KUKA KRL program: EPS_2_251806_MH09A_A_20260223023037.src

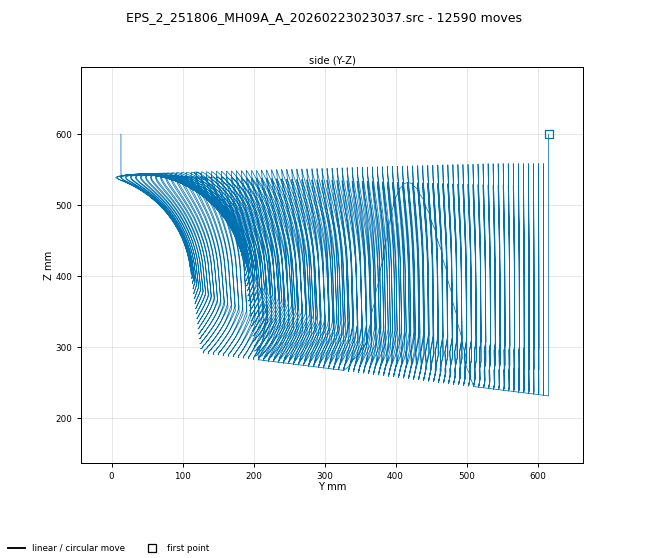
[picture p0: tool path of EPS_2_251806_MH09A_A_20260223023037.src, 12590 of 12592 moves have a stored position in this frame; points joined in program order, loops and branches not executed]
&ACCESS RVP
&REL 4
&COMMENT QRS 19112012
&PARAM EDITMASK = *
DEF PART()
EXT BAS (BAS_COMMAND :IN,REAL :IN )
INT I
BAS (#INITMOV,0 )

;KUKA QRS Post kuka4.cps  Date:22-06-2017 !

File_ID=3077

QRS_PRE_INIT()

;Init var - Until changes are made in qrs_pre_init
Outlet_Square_prg=0
Inlet_1_Square_prg=0
Inlet_2_Square_prg=0
Inlet_3_Square_prg=0
Inlet_4_Square_prg=0
Inlet_5_Square_prg=0

Outlet_1={X 0.000, Y 532.860, Z 433.000, B 0.000, E1 0.000 }
Inlet_1={X 0.000, Y 535.020, Z 403.000, B 0.000, E1 166.000 }
Outlet_1_type=251
Inlet_1_type=251
;QRS#1=Sidecore dimensions
;QRS#2=250-10" PVC SDR 35
;QRS#3=250-10" PVC SDR 35
;QRS#4=
;QRS#5=
;QRS#6=
;QRS#7=
;QRS#8=
;QRS#9=14M PSX
;QRS#10=14M PSX
;QRS#11=
;QRS#12=
;QRS#13=
;QRS#14=
;QRS#15=
;QRS#16=1220x127x838 2,75'
;QRS#17=EPS Height
;QRS#18=558,5
;QRS#19=*
;QRS#20= UPDATED VERSION 22-06-2017
;QRS#21=*
Outlet_Square=0100
Inlet_1_Square=0100
Inlet_2_Square=0
Inlet_3_Square=0
Inlet_4_Square=0
Inlet_5_Square=0
Mill_Square=1
Outlet_Square_Prg=205
Inlet_1_Square_prg=205

QRS_INIT()

$ADVANCE=5

; T1
PTP {E1 173.595,E2 173.595}
PTP {X 0,Y 615.506,A -85,B 0,C 180,E1 173.595,E2 173.595,E3 0,E4 0,E5 0,E6 0}
QRS_SPEED_INIT()
LIN {X 0,Y 615.506,Z 600,A -85,B 0,C 180,E1 173.595,E2 173.595,E3 0,E4 0,E5 0,E6 0} C_VEL
LIN {X 0,Y 615.506,Z 241.488,A -85,B 0,C 180,E1 173.595,E2 173.595} C_VEL
LIN {X 0,Y 615.506,Z 233.311,A -85,B 0,C 180,E1 173.595,E2 173.595} C_VEL
LIN {X 0,Y 615.49,Z 231.311,A -85,B 0,C 180,E1 173.408,E2 173.408} C_VEL
LIN {X 0,Y 615.485,Z 231.324,A -85,B 0,C 180,E1 170.802,E2 170.802} C_VEL
LIN {X 0,Y 615.466,Z 231.313,A -85,B 0,C 180,E1 168.14,E2 168.14} C_VEL
LIN {X 0,Y 615.489,Z 231.314,A -85,B 0,C 180,E1 165.452,E2 165.452} C_VEL
LIN {X 0,Y 615.469,Z 231.32,A -85,B 0,C 180,E1 162.73,E2 162.73} C_VEL
LIN {X 0,Y 615.486,Z 231.309,A -85,B 0,C 180,E1 159.968,E2 159.968} C_VEL
LIN {X 0,Y 615.488,Z 231.326,A -85,B 0,C 180,E1 157.157,E2 157.157} C_VEL
LIN {X 0,Y 615.46,Z 231.314,A -85,B 0,C 180,E1 154.434,E2 154.434} C_VEL
LIN {X 0,Y 615.49,Z 231.32,A -85,B 0,C 180,E1 151.547,E2 151.547} C_VEL
LIN {X 0,Y 615.462,Z 231.319,A -85,B 0,C 180,E1 148.916,E2 148.916} C_VEL
LIN {X 0,Y 615.464,Z 231.313,A -85,B 0,C 180,E1 146.467,E2 146.467} C_VEL
LIN {X 0,Y 615.485,Z 231.326,A -85,B 0,C 180,E1 143.577,E2 143.577} C_VEL
LIN {X 0,Y 615.456,Z 231.318,A -85,B 0,C 180,E1 140.94,E2 140.94} C_VEL
LIN {X 0,Y 615.467,Z 231.312,A -85,B 0,C 180,E1 138.526,E2 138.526} C_VEL
LIN {X 0,Y 615.494,Z 231.32,A -85,B 0,C 180,E1 135.853,E2 135.853} C_VEL
LIN {X 0,Y 615.458,Z 231.32,A -85,B 0,C 180,E1 133.246,E2 133.246} C_VEL
LIN {X 0,Y 615.47,Z 231.312,A -85,B 0,C 180,E1 130.607,E2 130.607} C_VEL
LIN {X 0,Y 615.49,Z 231.321,A -85,B 0,C 180,E1 128.015,E2 128.015} C_VEL
LIN {X 0,Y 615.467,Z 231.323,A -85,B 0,C 180,E1 125.616,E2 125.616} C_VEL
LIN {X 0,Y 615.48,Z 231.4,A -85,B 0,C 180,E1 124.594,E2 124.594} C_VEL
LIN {X 0,Y 615.442,Z 251.553,A -85,B 0,C 180,E1 121.687,E2 121.687} C_VEL
LIN {X 0,Y 615.455,Z 266.631,A -85,B 0,C 180,E1 119.539,E2 119.539} C_VEL
LIN {X 0,Y 615.471,Z 403.927,A -85,B 0,C 180,E1 117.892,E2 117.892} C_VEL
LIN {X 0,Y 615.484,Z 417.858,A -85,B 0,C 180,E1 117.591,E2 117.591} C_VEL
LIN {X 0,Y 615.487,Z 431.149,A -85,B 0,C 180,E1 117.176,E2 117.176} C_VEL
LIN {X 0,Y 615.488,Z 443.486,A -85,B 0,C 180,E1 116.67,E2 116.67} C_VEL
LIN {X 0,Y 615.485,Z 456.521,A -85,B 0,C 180,E1 115.988,E2 115.988} C_VEL
LIN {X 0,Y 615.497,Z 468.489,A -85,B 0,C 180,E1 115.209,E2 115.209} C_VEL
LIN {X 0,Y 615.499,Z 479.223,A -85,B 0,C 180,E1 114.361,E2 114.361} C_VEL
LIN {X 0,Y 615.497,Z 489.526,A -85,B 0,C 180,E1 113.377,E2 113.377} C_VEL
LIN {X 0,Y 615.492,Z 498.404,A -85,B 0,C 180,E1 112.351,E2 112.351} C_VEL
LIN {X 0,Y 615.494,Z 506.202,A -85,B 0,C 180,E1 111.255,E2 111.255} C_VEL
LIN {X 0,Y 615.495,Z 513.201,A -85,B 0,C 180,E1 110.032,E2 110.032} C_VEL
LIN {X 0,Y 615.492,Z 517.963,A -85,B 0,C 180,E1 108.991,E2 108.991} C_VEL
LIN {X 0,Y 615.495,Z 521.668,A -85,B 0,C 180,E1 107.956,E2 107.956} C_VEL
LIN {X 0,Y 615.493,Z 525.224,A -85,B 0,C 180,E1 106.586,E2 106.586} C_VEL
LIN {X 0,Y 615.493,Z 527.272,A -85,B 0,C 180,E1 105.225,E2 105.225} C_VEL
LIN {X 0,Y 615.497,Z 527.875,A -85,B 0,C 180,E1 103.874,E2 103.874} C_VEL
LIN {X 0,Y 615.489,Z 527.09,A -85,B 0,C 180,E1 102.53,E2 102.53} C_VEL
LIN {X 0,Y 615.491,Z 524.939,A -85,B 0,C 180,E1 101.193,E2 101.193} C_VEL
LIN {X 0,Y 615.499,Z 521.372,A -85,B 0,C 180,E1 99.862,E2 99.862} C_VEL
LIN {X 0,Y 615.494,Z 516.318,A -85,B 0,C 180,E1 98.536,E2 98.536} C_VEL
LIN {X 0,Y 615.495,Z 511.431,A -85,B 0,C 180,E1 97.545,E2 97.545} C_VEL
LIN {X 0,Y 615.497,Z 504.433,A -85,B 0,C 180,E1 96.392,E2 96.392} C_VEL
LIN {X 0,Y 615.497,Z 495.804,A -85,B 0,C 180,E1 95.241,E2 95.241} C_VEL
LIN {X 0,Y 615.497,Z 486.825,A -85,B 0,C 180,E1 94.256,E2 94.256} C_VEL
LIN {X 0,Y 615.497,Z 475.98,A -85,B 0,C 180,E1 93.273,E2 93.273} C_VEL
LIN {X 0,Y 615.498,Z 464.982,A -85,B 0,C 180,E1 92.454,E2 92.454} C_VEL
LIN {X 0,Y 615.491,Z 452.914,A -85,B 0,C 180,E1 91.718,E2 91.718} C_VEL
LIN {X 0,Y 615.494,Z 441.384,A -85,B 0,C 180,E1 91.145,E2 91.145} C_VEL
LIN {X 0,Y 615.492,Z 427.678,A -85,B 0,C 180,E1 90.613,E2 90.613} C_VEL
LIN {X 0,Y 615.47,Z 414.956,A -85,B 0,C 180,E1 90.245,E2 90.245} C_VEL
LIN {X 0,Y 615.453,Z 401.475,A -85,B 0,C 180,E1 89.979,E2 89.979} C_VEL
LIN {X 0,Y 615.447,Z 266.584,A -85,B 0,C 180,E1 88.364,E2 88.364} C_VEL
LIN {X 0,Y 615.484,Z 248.197,A -85,B 0,C 180,E1 85.744,E2 85.744} C_VEL
LIN {X 0,Y 615.489,Z 231.309,A -85,B 0,C 180,E1 83.293,E2 83.293} C_VEL
LIN {X 0,Y 615.476,Z 231.311,A -85,B 0,C 180,E1 80.801,E2 80.801} C_VEL
LIN {X 0,Y 615.487,Z 231.326,A -85,B 0,C 180,E1 78.139,E2 78.139} C_VEL
LIN {X 0,Y 615.484,Z 231.31,A -85,B 0,C 180,E1 75.451,E2 75.451} C_VEL
LIN {X 0,Y 615.472,Z 231.315,A -85,B 0,C 180,E1 72.729,E2 72.729} C_VEL
LIN {X 0,Y 615.485,Z 231.319,A -85,B 0,C 180,E1 69.968,E2 69.968} C_VEL
LIN {X 0,Y 615.479,Z 231.31,A -85,B 0,C 180,E1 67.156,E2 67.156} C_VEL
LIN {X 0,Y 615.496,Z 231.324,A -85,B 0,C 180,E1 64.285,E2 64.285} C_VEL
LIN {X 0,Y 615.483,Z 231.309,A -85,B 0,C 180,E1 61.342,E2 61.342} C_VEL
LIN {X 0,Y 615.474,Z 231.316,A -85,B 0,C 180,E1 58.913,E2 58.913} C_VEL
LIN {X 0,Y 615.498,Z 231.325,A -85,B 0,C 180,E1 56.462,E2 56.462} C_VEL
LIN {X 0,Y 615.485,Z 231.308,A -85,B 0,C 180,E1 53.576,E2 53.576} C_VEL
LIN {X 0,Y 615.477,Z 231.318,A -85,B 0,C 180,E1 50.937,E2 50.937} C_VEL
LIN {X 0,Y 615.493,Z 231.323,A -85,B 0,C 180,E1 48.528,E2 48.528} C_VEL
LIN {X 0,Y 615.492,Z 231.307,A -85,B 0,C 180,E1 45.852,E2 45.852} C_VEL
LIN {X 0,Y 615.479,Z 231.319,A -85,B 0,C 180,E1 43.048,E2 43.048} C_VEL
LIN {X 0,Y 615.483,Z 231.323,A -85,B 0,C 180,E1 40.605,E2 40.605} C_VEL
LIN {X 0,Y 615.484,Z 231.309,A -85,B 0,C 180,E1 38.013,E2 38.013} C_VEL
LIN {X 0,Y 615.479,Z 231.311,A -85,B 0,C 180,E1 35.615,E2 35.615} C_VEL
LIN {X 0,Y 615.479,Z 231.319,A -85,B 0,C 180,E1 33.235,E2 33.235} C_VEL
LIN {X 0,Y 615.489,Z 231.327,A -85,B 0,C 180,E1 30.918,E2 30.918} C_VEL
LIN {X 0,Y 615.479,Z 231.314,A -85,B 0,C 180,E1 28.451,E2 28.451} C_VEL
LIN {X 0,Y 615.478,Z 231.312,A -85,B 0,C 180,E1 25.715,E2 25.715} C_VEL
LIN {X 0,Y 615.475,Z 231.316,A -85,B 0,C 180,E1 23.556,E2 23.556} C_VEL
LIN {X 0,Y 615.479,Z 231.319,A -85,B 0,C 180,E1 21.431,E2 21.431} C_VEL
LIN {X 0,Y 615.477,Z 231.314,A -85,B 0,C 180,E1 18.605,E2 18.605} C_VEL
LIN {X 0,Y 615.476,Z 231.312,A -85,B 0,C 180,E1 15.904,E2 15.904} C_VEL
LIN {X 0,Y 615.494,Z 231.324,A -85,B 0,C 180,E1 13.2,E2 13.2} C_VEL
LIN {X 0,Y 615.486,Z 231.309,A -85,B 0,C 180,E1 10.526,E2 10.526} C_VEL
LIN {X 0,Y 615.477,Z 231.315,A -85,B 0,C 180,E1 7.875,E2 7.875} C_VEL
LIN {X 0,Y 615.487,Z 231.322,A -85,B 0,C 180,E1 5.24,E2 5.24} C_VEL
LIN {X 0,Y 615.488,Z 231.308,A -85,B 0,C 180,E1 2.617,E2 2.617} C_VEL
LIN {X 0,Y 615.478,Z 231.315,A -85,B 0,C 180,E1 -0.001,E2 -0.001} C_VEL
LIN {X 0,Y 615.486,Z 231.322,A -85,B 0,C 180,E1 -2.619,E2 -2.619} C_VEL
LIN {X 0,Y 615.487,Z 231.308,A -85,B 0,C 180,E1 -5.242,E2 -5.242} C_VEL
LIN {X 0,Y 615.479,Z 231.315,A -85,B 0,C 180,E1 -7.877,E2 -7.877} C_VEL
LIN {X 0,Y 615.484,Z 231.321,A -85,B 0,C 180,E1 -10.528,E2 -10.528} C_VEL
LIN {X 0,Y 615.493,Z 231.306,A -85,B 0,C 180,E1 -13.202,E2 -13.202} C_VEL
LIN {X 0,Y 615.482,Z 231.319,A -85,B 0,C 180,E1 -15.906,E2 -15.906} C_VEL
LIN {X 0,Y 615.475,Z 231.316,A -85,B 0,C 180,E1 -18.647,E2 -18.647} C_VEL
LIN {X 0,Y 615.479,Z 231.312,A -85,B 0,C 180,E1 -21.433,E2 -21.433} C_VEL
LIN {X 0,Y 615.483,Z 231.321,A -85,B 0,C 180,E1 -24.273,E2 -24.273} C_VEL
LIN {X 0,Y 615.491,Z 231.307,A -85,B 0,C 180,E1 -27.178,E2 -27.178} C_VEL
LIN {X 0,Y 615.483,Z 231.321,A -85,B 0,C 180,E1 -30.161,E2 -30.161} C_VEL
LIN {X 0,Y 615.473,Z 231.315,A -85,B 0,C 180,E1 -32.459,E2 -32.459} C_VEL
LIN {X 0,Y 615.49,Z 231.307,A -85,B 0,C 180,E1 -34.815,E2 -34.815} C_VEL
LIN {X 0,Y 615.482,Z 231.313,A -85,B 0,C 180,E1 -37.243,E2 -37.243} C_VEL
LIN {X 0,Y 615.474,Z 231.32,A -85,B 0,C 180,E1 -40.089,E2 -40.089} C_VEL
LIN {X 0,Y 615.473,Z 231.313,A -85,B 0,C 180,E1 -42.355,E2 -42.355} C_VEL
LIN {X 0,Y 615.483,Z 231.312,A -85,B 0,C 180,E1 -45.069,E2 -45.069} C_VEL
LIN {X 0,Y 615.496,Z 231.325,A -85,B 0,C 180,E1 -47.649,E2 -47.649} C_VEL
LIN {X 0,Y 615.474,Z 231.313,A -85,B 0,C 180,E1 -50.25,E2 -50.25} C_VEL
LIN {X 0,Y 615.479,Z 231.315,A -85,B 0,C 180,E1 -53.065,E2 -53.065} C_VEL
LIN {X 0,Y 615.489,Z 231.321,A -85,B 0,C 180,E1 -55.3,E2 -55.3} C_VEL
LIN {X 0,Y 615.482,Z 231.321,A -85,B 0,C 180,E1 -57.671,E2 -57.671} C_VEL
LIN {X 0,Y 615.493,Z 231.307,A -85,B 0,C 180,E1 -60.595,E2 -60.595} C_VEL
LIN {X 0,Y 615.48,Z 231.321,A -85,B 0,C 180,E1 -63.556,E2 -63.556} C_VEL
LIN {X 0,Y 615.486,Z 231.309,A -85,B 0,C 180,E1 -66.444,E2 -66.444} C_VEL
LIN {X 0,Y 615.486,Z 231.548,A -85,B 0,C 180,E1 -66.533,E2 -66.533} C_VEL
LIN {X 0,Y 615.487,Z 254.856,A -85,B 0,C 180,E1 -69.444,E2 -69.444} C_VEL
LIN {X 0,Y 615.493,Z 277.448,A -85,B 0,C 180,E1 -72.215,E2 -72.215} C_VEL
LIN {X 0,Y 615.49,Z 295.428,A -85,B 0,C 180,E1 -74.393,E2 -74.393} C_VEL
LIN {X 0,Y 615.488,Z 433.076,A -85,B 0,C 180,E1 -76.048,E2 -76.048} C_VEL
LIN {X 0,Y 615.494,Z 446.865,A -85,B 0,C 180,E1 -76.337,E2 -76.337} C_VEL
LIN {X 0,Y 615.487,Z 460.574,A -85,B 0,C 180,E1 -76.757,E2 -76.757} C_VEL
LIN {X 0,Y 615.497,Z 473.841,A -85,B 0,C 180,E1 -77.303,E2 -77.303} C_VEL
LIN {X 0,Y 615.483,Z 486.604,A -85,B 0,C 180,E1 -77.972,E2 -77.972} C_VEL
LIN {X 0,Y 615.499,Z 499.342,A -85,B 0,C 180,E1 -78.807,E2 -78.807} C_VEL
LIN {X 0,Y 615.498,Z 509.75,A -85,B 0,C 180,E1 -79.64,E2 -79.64} C_VEL
LIN {X 0,Y 615.496,Z 520.089,A -85,B 0,C 180,E1 -80.636,E2 -80.636} C_VEL
LIN {X 0,Y 615.497,Z 528.603,A -85,B 0,C 180,E1 -81.629,E2 -81.629} C_VEL
LIN {X 0,Y 615.496,Z 536.727,A -85,B 0,C 180,E1 -82.785,E2 -82.785} C_VEL
LIN {X 0,Y 615.496,Z 542.43,A -85,B 0,C 180,E1 -83.773,E2 -83.773} C_VEL
LIN {X 0,Y 615.495,Z 547.08,A -85,B 0,C 180,E1 -84.759,E2 -84.759} C_VEL
LIN {X 0,Y 615.494,Z 551.902,A -85,B 0,C 180,E1 -86.072,E2 -86.072} C_VEL
LIN {X 0,Y 615.496,Z 555.252,A -85,B 0,C 180,E1 -87.382,E2 -87.382} C_VEL
LIN {X 0,Y 615.489,Z 557.229,A -85,B 0,C 180,E1 -88.691,E2 -88.691} C_VEL
LIN {X 0,Y 615.493,Z 557.889,A -85,B 0,C 180,E1 -90,E2 -90} C_VEL
LIN {X 0,Y 615.489,Z 557.229,A -85,B 0,C 180,E1 -91.308,E2 -91.308} C_VEL
LIN {X 0,Y 615.496,Z 555.252,A -85,B 0,C 180,E1 -92.618,E2 -92.618} C_VEL
LIN {X 0,Y 615.494,Z 551.902,A -85,B 0,C 180,E1 -93.928,E2 -93.928} C_VEL
LIN {X 0,Y 615.495,Z 547.081,A -85,B 0,C 180,E1 -95.241,E2 -95.241} C_VEL
LIN {X 0,Y 615.496,Z 540.629,A -85,B 0,C 180,E1 -96.556,E2 -96.556} C_VEL
LIN {X 0,Y 615.497,Z 533.442,A -85,B 0,C 180,E1 -97.71,E2 -97.71} C_VEL
LIN {X 0,Y 615.498,Z 525.905,A -85,B 0,C 180,E1 -98.702,E2 -98.702} C_VEL
LIN {X 0,Y 615.496,Z 516.855,A -85,B 0,C 180,E1 -99.696,E2 -99.696} C_VEL
LIN {X 0,Y 615.498,Z 506.76,A -85,B 0,C 180,E1 -100.618,E2 -100.618} C_VEL
LIN {X 0,Y 615.498,Z 495.862,A -85,B 0,C 180,E1 -101.443,E2 -101.443} C_VEL
LIN {X 0,Y 615.484,Z 483.712,A -85,B 0,C 180,E1 -102.195,E2 -102.195} C_VEL
LIN {X 0,Y 615.493,Z 470.098,A -85,B 0,C 180,E1 -102.865,E2 -102.865} C_VEL
LIN {X 0,Y 615.49,Z 456.845,A -85,B 0,C 180,E1 -103.369,E2 -103.369} C_VEL
LIN {X 0,Y 615.493,Z 443.301,A -85,B 0,C 180,E1 -103.747,E2 -103.747} C_VEL
LIN {X 0,Y 615.485,Z 428.996,A -85,B 0,C 180,E1 -104.009,E2 -104.009} C_VEL
LIN {X 0,Y 615.49,Z 295.43,A -85,B 0,C 180,E1 -105.607,E2 -105.607} C_VEL
LIN {X 0,Y 615.483,Z 273.41,A -85,B 0,C 180,E1 -108.277,E2 -108.277} C_VEL
LIN {X 0,Y 615.469,Z 252.038,A -85,B 0,C 180,E1 -110.906,E2 -110.906} C_VEL
LIN {X 0,Y 615.485,Z 231.309,A -85,B 0,C 180,E1 -113.511,E2 -113.511} C_VEL
LIN {X 0,Y 615.485,Z 231.308,A -85,B 0,C 180,E1 -115.715,E2 -115.715} C_VEL
LIN {X 0,Y 615.485,Z 231.327,A -85,B 0,C 180,E1 -118.657,E2 -118.657} C_VEL
LIN {X 0,Y 615.481,Z 231.314,A -85,B 0,C 180,E1 -121.085,E2 -121.085} C_VEL
LIN {X 0,Y 615.492,Z 231.307,A -85,B 0,C 180,E1 -123.534,E2 -123.534} C_VEL
LIN {X 0,Y 615.484,Z 231.328,A -85,B 0,C 180,E1 -126.424,E2 -126.424} C_VEL
LIN {X 0,Y 615.483,Z 231.311,A -85,B 0,C 180,E1 -129.061,E2 -129.061} C_VEL
LIN {X 0,Y 615.486,Z 231.308,A -85,B 0,C 180,E1 -131.473,E2 -131.473} C_VEL
LIN {X 0,Y 615.49,Z 231.323,A -85,B 0,C 180,E1 -134.148,E2 -134.148} C_VEL
LIN {X 0,Y 615.483,Z 231.31,A -85,B 0,C 180,E1 -136.952,E2 -136.952} C_VEL
LIN {X 0,Y 615.482,Z 231.31,A -85,B 0,C 180,E1 -139.393,E2 -139.393} C_VEL
LIN {X 0,Y 615.483,Z 231.324,A -85,B 0,C 180,E1 -141.987,E2 -141.987} C_VEL
LIN {X 0,Y 615.479,Z 231.319,A -85,B 0,C 180,E1 -144.383,E2 -144.383} C_VEL
LIN {X 0,Y 615.48,Z 231.31,A -85,B 0,C 180,E1 -146.763,E2 -146.763} C_VEL
LIN {X 0,Y 615.487,Z 231.308,A -85,B 0,C 180,E1 -149.08,E2 -149.08} C_VEL
LIN {X 0,Y 615.48,Z 231.318,A -85,B 0,C 180,E1 -151.549,E2 -151.549} C_VEL
LIN {X 0,Y 615.473,Z 231.317,A -85,B 0,C 180,E1 -154.283,E2 -154.283} C_VEL
LIN {X 0,Y 615.472,Z 231.314,A -85,B 0,C 180,E1 -156.442,E2 -156.442} C_VEL
LIN {X 0,Y 615.483,Z 231.315,A -85,B 0,C 180,E1 -159.268,E2 -159.268} C_VEL
LIN {X 0,Y 615.475,Z 231.319,A -85,B 0,C 180,E1 -162.042,E2 -162.042} C_VEL
LIN {X 0,Y 615.49,Z 231.308,A -85,B 0,C 180,E1 -164.773,E2 -164.773} C_VEL
LIN {X 0,Y 615.486,Z 231.325,A -85,B 0,C 180,E1 -167.469,E2 -167.469} C_VEL
LIN {X 0,Y 615.47,Z 231.314,A -85,B 0,C 180,E1 -170.137,E2 -170.137} C_VEL
LIN {X 0,Y 615.487,Z 231.31,A -85,B 0,C 180,E1 -172.784,E2 -172.784} C_VEL
LIN {X 0,Y 615.496,Z 231.325,A -85,B 0,C 180,E1 -175.415,E2 -175.415} C_VEL
LIN {X 0,Y 615.468,Z 231.314,A -85,B 0,C 180,E1 -178.036,E2 -178.036} C_VEL
LIN {X 0,Y 615.486,Z 231.311,A -85,B 0,C 180,E1 -180.653,E2 -180.653} C_VEL
LIN {X 0,Y 615.488,Z 231.325,A -85,B 0,C 180,E1 -183.272,E2 -183.272} C_VEL
LIN {X 0,Y 615.466,Z 231.314,A -85,B 0,C 180,E1 -185.898,E2 -185.898} C_VEL
LIN {X 0,Y 615.49,Z 231.311,A -85,B 0,C 180,E1 -186.592,E2 -186.592} C_VEL
LIN {X 0,Y 614.813,Z 231.47,A -85,B 0,C 180,E1 -187.138,E2 -187.138} C_VEL
LIN {X 0,Y 611.977,Z 231.873,A -85,B 0,C 180,E1 -188.024,E2 -188.024} C_VEL
LIN {X 0,Y 609.583,Z 232.188,A -85,B 0,C 180,E1 -188.736,E2 -188.736} C_VEL
LIN {X 0,Y 608.543,Z 232.308,A -85,B 0,C 180,E1 -189.286,E2 -189.286} C_VEL
LIN {X 0,Y 608.451,Z 232.317,A -85,B 0,C 180,E1 -189.472,E2 -189.472} C_VEL
LIN {X 0,Y 608.447,Z 232.313,A -85,B 0,C 180,E1 -191.999,E2 -191.999} C_VEL
LIN {X 0,Y 608.472,Z 232.316,A -85,B 0,C 180,E1 -194.719,E2 -194.719} C_VEL
LIN {X 0,Y 608.437,Z 232.316,A -85,B 0,C 180,E1 -197.476,E2 -197.476} C_VEL
LIN {X 0,Y 608.462,Z 232.313,A -85,B 0,C 180,E1 -200.273,E2 -200.273} C_VEL
LIN {X 0,Y 608.441,Z 232.319,A -85,B 0,C 180,E1 -203.123,E2 -203.123} C_VEL
LIN {X 0,Y 608.451,Z 232.313,A -85,B 0,C 180,E1 -205.72,E2 -205.72} C_VEL
LIN {X 0,Y 608.473,Z 232.32,A -85,B 0,C 180,E1 -208.622,E2 -208.622} C_VEL
LIN {X 0,Y 608.429,Z 232.316,A -85,B 0,C 180,E1 -211.317,E2 -211.317} C_VEL
LIN {X 0,Y 608.459,Z 232.312,A -85,B 0,C 180,E1 -213.735,E2 -213.735} C_VEL
LIN {X 0,Y 608.467,Z 232.314,A -85,B 0,C 180,E1 -216.089,E2 -216.089} C_VEL
LIN {X 0,Y 608.454,Z 232.32,A -85,B 0,C 180,E1 -218.587,E2 -218.587} C_VEL
LIN {X 0,Y 608.438,Z 232.314,A -85,B 0,C 180,E1 -221.341,E2 -221.341} C_VEL
LIN {X 0,Y 608.47,Z 232.314,A -85,B 0,C 180,E1 -223.867,E2 -223.867} C_VEL
LIN {X 0,Y 608.448,Z 232.317,A -85,B 0,C 180,E1 -226.691,E2 -226.691} C_VEL
LIN {X 0,Y 608.425,Z 232.318,A -85,B 0,C 180,E1 -228.822,E2 -228.822} C_VEL
LIN {X 0,Y 608.451,Z 232.314,A -85,B 0,C 180,E1 -231.412,E2 -231.412} C_VEL
LIN {X 0,Y 608.468,Z 232.319,A -85,B 0,C 180,E1 -233.949,E2 -233.949} C_VEL
LIN {X 0,Y 608.485,Z 232.486,A -85,B 0,C 180,E1 -235.316,E2 -235.316} C_VEL
LIN {X 0,Y 608.489,Z 250.245,A -85,B 0,C 180,E1 -237.908,E2 -237.908} C_VEL
LIN {X 0,Y 608.446,Z 266.656,A -85,B 0,C 180,E1 -240.268,E2 -240.268} C_VEL
LIN {X 0,Y 608.63,Z 273.911,A -85,B 0,C 180,E1 -240.373,E2 -240.373} C_VEL
LIN {X 0,Y 608.6,Z 402.894,A -85,B 0,C 180,E1 -241.929,E2 -241.929} C_VEL
LIN {X 0,Y 608.572,Z 417.186,A -85,B 0,C 180,E1 -242.232,E2 -242.232} C_VEL
LIN {X 0,Y 608.573,Z 431.379,A -85,B 0,C 180,E1 -242.679,E2 -242.679} C_VEL
LIN {X 0,Y 608.544,Z 444.524,A -85,B 0,C 180,E1 -243.231,E2 -243.231} C_VEL
LIN {X 0,Y 608.53,Z 456.673,A -85,B 0,C 180,E1 -243.877,E2 -243.877} C_VEL
LIN {X 0,Y 608.498,Z 469.197,A -85,B 0,C 180,E1 -244.702,E2 -244.702} C_VEL
LIN {X 0,Y 608.486,Z 479.815,A -85,B 0,C 180,E1 -245.554,E2 -245.554} C_VEL
LIN {X 0,Y 608.483,Z 489.811,A -85,B 0,C 180,E1 -246.518,E2 -246.518} C_VEL
LIN {X 0,Y 608.46,Z 499.058,A -85,B 0,C 180,E1 -247.595,E2 -247.595} C_VEL
LIN {X 0,Y 608.459,Z 506.609,A -85,B 0,C 180,E1 -248.664,E2 -248.664} C_VEL
LIN {X 0,Y 608.441,Z 512.759,A -85,B 0,C 180,E1 -249.726,E2 -249.726} C_VEL
LIN {X 0,Y 608.434,Z 517.727,A -85,B 0,C 180,E1 -250.78,E2 -250.78} C_VEL
LIN {X 0,Y 608.448,Z 522.778,A -85,B 0,C 180,E1 -252.177,E2 -252.177} C_VEL
LIN {X 0,Y 608.419,Z 526.013,A -85,B 0,C 180,E1 -253.481,E2 -253.481} C_VEL
LIN {X 0,Y 608.415,Z 527.679,A -85,B 0,C 180,E1 -254.593,E2 -254.593} C_VEL
LIN {X 0,Y 608.428,Z 528.494,A -85,B 0,C 180,E1 -255.992,E2 -255.992} C_VEL
LIN {X 0,Y 608.414,Z 527.884,A -85,B 0,C 180,E1 -257.322,E2 -257.322} C_VEL
LIN {X 0,Y 608.417,Z 525.87,A -85,B 0,C 180,E1 -258.675,E2 -258.675} C_VEL
LIN {X 0,Y 608.433,Z 522.43,A -85,B 0,C 180,E1 -260.023,E2 -260.023} C_VEL
LIN {X 0,Y 608.426,Z 517.496,A -85,B 0,C 180,E1 -261.364,E2 -261.364} C_VEL
LIN {X 0,Y 608.445,Z 512.745,A -85,B 0,C 180,E1 -262.367,E2 -262.367} C_VEL
LIN {X 0,Y 608.455,Z 505.374,A -85,B 0,C 180,E1 -263.61,E2 -263.61} C_VEL
LIN {X 0,Y 608.461,Z 497.416,A -85,B 0,C 180,E1 -264.698,E2 -264.698} C_VEL
LIN {X 0,Y 608.48,Z 488.625,A -85,B 0,C 180,E1 -265.695,E2 -265.695} C_VEL
LIN {X 0,Y 608.491,Z 478.048,A -85,B 0,C 180,E1 -266.69,E2 -266.69} C_VEL
LIN {X 0,Y 608.514,Z 466.264,A -85,B 0,C 180,E1 -267.601,E2 -267.601} C_VEL
LIN {X 0,Y 608.526,Z 454.439,A -85,B 0,C 180,E1 -268.346,E2 -268.346} C_VEL
LIN {X 0,Y 608.558,Z 441.332,A -85,B 0,C 180,E1 -269.008,E2 -269.008} C_VEL
LIN {X 0,Y 608.575,Z 427.573,A -85,B 0,C 180,E1 -269.545,E2 -269.545} C_VEL
LIN {X 0,Y 608.588,Z 413.878,A -85,B 0,C 180,E1 -269.938,E2 -269.938} C_VEL
LIN {X 0,Y 608.581,Z 399.69,A -85,B 0,C 180,E1 -270.207,E2 -270.207} C_VEL
LIN {X 0,Y 608.518,Z 267.308,A -85,B 0,C 180,E1 -271.799,E2 -271.799} C_VEL
LIN {X 0,Y 608.44,Z 266.67,A -85,B 0,C 180,E1 -271.82,E2 -271.82} C_VEL
LIN {X 0,Y 608.519,Z 248.244,A -85,B 0,C 180,E1 -274.471,E2 -274.471} C_VEL
LIN {X 0,Y 608.484,Z 232.31,A -85,B 0,C 180,E1 -276.805,E2 -276.805} C_VEL
LIN {X 0,Y 608.461,Z 232.313,A -85,B 0,C 180,E1 -279.306,E2 -279.306} C_VEL
LIN {X 0,Y 608.46,Z 232.321,A -85,B 0,C 180,E1 -282,E2 -282} C_VEL
LIN {X 0,Y 608.468,Z 232.311,A -85,B 0,C 180,E1 -284.72,E2 -284.72} C_VEL
LIN {X 0,Y 608.444,Z 232.318,A -85,B 0,C 180,E1 -287.477,E2 -287.477} C_VEL
LIN {X 0,Y 608.461,Z 232.314,A -85,B 0,C 180,E1 -290.274,E2 -290.274} C_VEL
LIN {X 0,Y 608.444,Z 232.315,A -85,B 0,C 180,E1 -293.124,E2 -293.124} C_VEL
LIN {X 0,Y 608.475,Z 232.319,A -85,B 0,C 180,E1 -295.725,E2 -295.725} C_VEL
LIN {X 0,Y 608.471,Z 232.31,A -85,B 0,C 180,E1 -298.623,E2 -298.623} C_VEL
LIN {X 0,Y 608.465,Z 232.317,A -85,B 0,C 180,E1 -301.316,E2 -301.316} C_VEL
LIN {X 0,Y 608.477,Z 232.316,A -85,B 0,C 180,E1 -303.738,E2 -303.738} C_VEL
LIN {X 0,Y 608.466,Z 232.312,A -85,B 0,C 180,E1 -306.09,E2 -306.09} C_VEL
LIN {X 0,Y 608.459,Z 232.312,A -85,B 0,C 180,E1 -308.588,E2 -308.588} C_VEL
LIN {X 0,Y 608.462,Z 232.322,A -85,B 0,C 180,E1 -311.344,E2 -311.344} C_VEL
LIN {X 0,Y 608.457,Z 232.312,A -85,B 0,C 180,E1 -314.266,E2 -314.266} C_VEL
LIN {X 0,Y 608.446,Z 232.32,A -85,B 0,C 180,E1 -317.041,E2 -317.041} C_VEL
LIN {X 0,Y 608.448,Z 232.316,A -85,B 0,C 180,E1 -319.698,E2 -319.698} C_VEL
LIN {X 0,Y 608.464,Z 232.311,A -85,B 0,C 180,E1 -322.255,E2 -322.255} C_VEL
LIN {X 0,Y 608.481,Z 232.319,A -85,B 0,C 180,E1 -325.089,E2 -325.089} C_VEL
LIN {X 0,Y 608.458,Z 232.312,A -85,B 0,C 180,E1 -327.907,E2 -327.907} C_VEL
LIN {X 0,Y 608.468,Z 232.311,A -85,B 0,C 180,E1 -330.222,E2 -330.222} C_VEL
LIN {X 0,Y 608.479,Z 232.316,A -85,B 0,C 180,E1 -332.79,E2 -332.79} C_VEL
LIN {X 0,Y 608.481,Z 232.309,A -85,B 0,C 180,E1 -335.844,E2 -335.844} C_VEL
LIN {X 0,Y 608.466,Z 232.313,A -85,B 0,C 180,E1 -338.31,E2 -338.31} C_VEL
LIN {X 0,Y 608.447,Z 232.319,A -85,B 0,C 180,E1 -341.131,E2 -341.131} C_VEL
LIN {X 0,Y 608.454,Z 232.312,A -85,B 0,C 180,E1 -343.907,E2 -343.907} C_VEL
LIN {X 0,Y 608.467,Z 232.32,A -85,B 0,C 180,E1 -346.645,E2 -346.645} C_VEL
LIN {X 0,Y 608.461,Z 232.313,A -85,B 0,C 180,E1 -349.351,E2 -349.351} C_VEL
LIN {X 0,Y 608.469,Z 232.312,A -85,B 0,C 180,E1 -352.034,E2 -352.034} C_VEL
LIN {X 0,Y 608.465,Z 232.32,A -85,B 0,C 180,E1 -354.699,E2 -354.699} C_VEL
LIN {X 0,Y 608.478,Z 232.31,A -85,B 0,C 180,E1 -357.353,E2 -357.353} C_VEL
LIN {X 0,Y 608.469,Z 232.313,A -85,B 0,C 180,E1 -360.001,E2 -360.001} C_VEL
LIN {X 0,Y 608.477,Z 232.316,A -85,B 0,C 180,E1 -362.649,E2 -362.649} C_VEL
LIN {X 0,Y 608.465,Z 232.311,A -85,B 0,C 180,E1 -365.303,E2 -365.303} C_VEL
LIN {X 0,Y 608.47,Z 232.314,A -85,B 0,C 180,E1 -367.968,E2 -367.968} C_VEL
LIN {X 0,Y 608.46,Z 232.316,A -85,B 0,C 180,E1 -370.651,E2 -370.651} C_VEL
LIN {X 0,Y 608.467,Z 232.311,A -85,B 0,C 180,E1 -373.357,E2 -373.357} C_VEL
LIN {X 0,Y 608.457,Z 232.321,A -85,B 0,C 180,E1 -376.095,E2 -376.095} C_VEL
LIN {X 0,Y 608.449,Z 232.314,A -85,B 0,C 180,E1 -378.87,E2 -378.87} C_VEL
LIN {X 0,Y 608.468,Z 232.314,A -85,B 0,C 180,E1 -381.692,E2 -381.692} C_VEL
LIN {X 0,Y 608.453,Z 232.315,A -85,B 0,C 180,E1 -384.572,E2 -384.572} C_VEL
LIN {X 0,Y 608.483,Z 232.309,A -85,B 0,C 180,E1 -387.21,E2 -387.21} C_VEL
LIN {X 0,Y 608.468,Z 232.321,A -85,B 0,C 180,E1 -389.974,E2 -389.974} C_VEL
LIN {X 0,Y 608.45,Z 232.314,A -85,B 0,C 180,E1 -392.522,E2 -392.522} C_VEL
LIN {X 0,Y 608.443,Z 232.316,A -85,B 0,C 180,E1 -395.278,E2 -395.278} C_VEL
LIN {X 0,Y 608.466,Z 232.321,A -85,B 0,C 180,E1 -397.747,E2 -397.747} C_VEL
LIN {X 0,Y 608.442,Z 232.316,A -85,B 0,C 180,E1 -400.329,E2 -400.329} C_VEL
LIN {X 0,Y 608.469,Z 232.314,A -85,B 0,C 180,E1 -403.31,E2 -403.31} C_VEL
LIN {X 0,Y 608.464,Z 232.314,A -85,B 0,C 180,E1 -406.131,E2 -406.131} C_VEL
LIN {X 0,Y 608.456,Z 232.312,A -85,B 0,C 180,E1 -408.825,E2 -408.825} C_VEL
LIN {X 0,Y 608.459,Z 232.318,A -85,B 0,C 180,E1 -411.761,E2 -411.761} C_VEL
LIN {X 0,Y 608.443,Z 232.317,A -85,B 0,C 180,E1 -413.955,E2 -413.955} C_VEL
LIN {X 0,Y 608.463,Z 232.311,A -85,B 0,C 180,E1 -416.33,E2 -416.33} C_VEL
LIN {X 0,Y 608.447,Z 232.314,A -85,B 0,C 180,E1 -418.733,E2 -418.733} C_VEL
LIN {X 0,Y 608.472,Z 232.321,A -85,B 0,C 180,E1 -421.381,E2 -421.381} C_VEL
LIN {X 0,Y 608.474,Z 232.31,A -85,B 0,C 180,E1 -424.279,E2 -424.279} C_VEL
LIN {X 0,Y 608.485,Z 232.431,A -85,B 0,C 180,E1 -426.36,E2 -426.36} C_VEL
LIN {X 0,Y 608.589,Z 249.21,A -85,B 0,C 180,E1 -428.491,E2 -428.491} C_VEL
LIN {X 0,Y 608.533,Z 271.49,A -85,B 0,C 180,E1 -431.267,E2 -431.267} C_VEL
LIN {X 0,Y 608.521,Z 294.428,A -85,B 0,C 180,E1 -434.08,E2 -434.08} C_VEL
LIN {X 0,Y 608.515,Z 295.576,A -85,B 0,C 180,E1 -434.22,E2 -434.22} C_VEL
LIN {X 0,Y 608.6,Z 433.465,A -85,B 0,C 180,E1 -435.894,E2 -435.894} C_VEL
LIN {X 0,Y 608.592,Z 447.633,A -85,B 0,C 180,E1 -436.2,E2 -436.2} C_VEL
LIN {X 0,Y 608.578,Z 461.716,A -85,B 0,C 180,E1 -436.646,E2 -436.646} C_VEL
LIN {X 0,Y 608.561,Z 473.887,A -85,B 0,C 180,E1 -437.155,E2 -437.155} C_VEL
LIN {X 0,Y 608.511,Z 486.683,A -85,B 0,C 180,E1 -437.832,E2 -437.832} C_VEL
LIN {X 0,Y 608.499,Z 499.473,A -85,B 0,C 180,E1 -438.677,E2 -438.677} C_VEL
LIN {X 0,Y 608.496,Z 509.933,A -85,B 0,C 180,E1 -439.519,E2 -439.519} C_VEL
LIN {X 0,Y 608.479,Z 520.335,A -85,B 0,C 180,E1 -440.527,E2 -440.527} C_VEL
LIN {X 0,Y 608.464,Z 528.915,A -85,B 0,C 180,E1 -441.532,E2 -441.532} C_VEL
LIN {X 0,Y 608.461,Z 537.114,A -85,B 0,C 180,E1 -442.701,E2 -442.701} C_VEL
LIN {X 0,Y 608.444,Z 543.546,A -85,B 0,C 180,E1 -443.831,E2 -443.831} C_VEL
LIN {X 0,Y 608.437,Z 548.962,A -85,B 0,C 180,E1 -445.03,E2 -445.03} C_VEL
LIN {X 0,Y 608.431,Z 552.441,A -85,B 0,C 180,E1 -446.026,E2 -446.026} C_VEL
LIN {X 0,Y 608.424,Z 555.831,A -85,B 0,C 180,E1 -447.352,E2 -447.352} C_VEL
LIN {X 0,Y 608.442,Z 557.83,A -85,B 0,C 180,E1 -448.676,E2 -448.676} C_VEL
LIN {X 0,Y 608.433,Z 558.5,A -85,B 0,C 180,E1 -450,E2 -450} C_VEL
LIN {X 0,Y 608.442,Z 557.831,A -85,B 0,C 180,E1 -451.324,E2 -451.324} C_VEL
LIN {X 0,Y 608.424,Z 555.831,A -85,B 0,C 180,E1 -452.648,E2 -452.648} C_VEL
LIN {X 0,Y 608.431,Z 552.442,A -85,B 0,C 180,E1 -453.974,E2 -453.974} C_VEL
LIN {X 0,Y 608.44,Z 547.568,A -85,B 0,C 180,E1 -455.302,E2 -455.302} C_VEL
LIN {X 0,Y 608.445,Z 541.212,A -85,B 0,C 180,E1 -456.603,E2 -456.603} C_VEL
LIN {X 0,Y 608.453,Z 533.799,A -85,B 0,C 180,E1 -457.8,E2 -457.8} C_VEL
LIN {X 0,Y 608.473,Z 524.825,A -85,B 0,C 180,E1 -458.97,E2 -458.97} C_VEL
LIN {X 0,Y 608.473,Z 515.394,A -85,B 0,C 180,E1 -459.977,E2 -459.977} C_VEL
LIN {X 0,Y 608.506,Z 504.049,A -85,B 0,C 180,E1 -460.973,E2 -460.973} C_VEL
LIN {X 0,Y 608.53,Z 492.153,A -85,B 0,C 180,E1 -461.829,E2 -461.829} C_VEL
LIN {X 0,Y 608.53,Z 479.078,A -85,B 0,C 180,E1 -462.591,E2 -462.591} C_VEL
LIN {X 0,Y 608.553,Z 466.18,A -85,B 0,C 180,E1 -463.184,E2 -463.184} C_VEL
LIN {X 0,Y 608.593,Z 452.193,A -85,B 0,C 180,E1 -463.672,E2 -463.672} C_VEL
LIN {X 0,Y 608.622,Z 438.471,A -85,B 0,C 180,E1 -464.012,E2 -464.012} C_VEL
LIN {X 0,Y 608.619,Z 422.194,A -85,B 0,C 180,E1 -464.257,E2 -464.257} C_VEL
LIN {X 0,Y 608.528,Z 295.577,A -85,B 0,C 180,E1 -465.78,E2 -465.78} C_VEL
LIN {X 0,Y 608.537,Z 273.426,A -85,B 0,C 180,E1 -468.493,E2 -468.493} C_VEL
LIN {X 0,Y 608.581,Z 252.038,A -85,B 0,C 180,E1 -471.154,E2 -471.154} C_VEL
LIN {X 0,Y 608.58,Z 232.962,A -85,B 0,C 180,E1 -473.569,E2 -473.569} C_VEL
LIN {X 0,Y 608.454,Z 232.314,A -85,B 0,C 180,E1 -473.664,E2 -473.664} C_VEL
LIN {X 0,Y 608.441,Z 232.316,A -85,B 0,C 180,E1 -476.035,E2 -476.035} C_VEL
LIN {X 0,Y 608.472,Z 232.321,A -85,B 0,C 180,E1 -478.619,E2 -478.619} C_VEL
LIN {X 0,Y 608.459,Z 232.313,A -85,B 0,C 180,E1 -481.316,E2 -481.316} C_VEL
LIN {X 0,Y 608.473,Z 232.311,A -85,B 0,C 180,E1 -483.734,E2 -483.734} C_VEL
LIN {X 0,Y 608.443,Z 232.318,A -85,B 0,C 180,E1 -486.091,E2 -486.091} C_VEL
LIN {X 0,Y 608.463,Z 232.319,A -85,B 0,C 180,E1 -488.587,E2 -488.587} C_VEL
LIN {X 0,Y 608.462,Z 232.311,A -85,B 0,C 180,E1 -491.342,E2 -491.342} C_VEL
LIN {X 0,Y 608.458,Z 232.323,A -85,B 0,C 180,E1 -494.264,E2 -494.264} C_VEL
LIN {X 0,Y 608.449,Z 232.313,A -85,B 0,C 180,E1 -497.039,E2 -497.039} C_VEL
LIN {X 0,Y 608.447,Z 232.316,A -85,B 0,C 180,E1 -499.696,E2 -499.696} C_VEL
LIN {X 0,Y 608.465,Z 232.319,A -85,B 0,C 180,E1 -502.253,E2 -502.253} C_VEL
LIN {X 0,Y 608.48,Z 232.309,A -85,B 0,C 180,E1 -505.088,E2 -505.088} C_VEL
LIN {X 0,Y 608.461,Z 232.321,A -85,B 0,C 180,E1 -507.905,E2 -507.905} C_VEL
LIN {X 0,Y 608.463,Z 232.317,A -85,B 0,C 180,E1 -510.22,E2 -510.22} C_VEL
LIN {X 0,Y 608.482,Z 232.309,A -85,B 0,C 180,E1 -512.79,E2 -512.79} C_VEL
LIN {X 0,Y 608.478,Z 232.319,A -85,B 0,C 180,E1 -515.844,E2 -515.844} C_VEL
LIN {X 0,Y 608.462,Z 232.313,A -85,B 0,C 180,E1 -518.308,E2 -518.308} C_VEL
LIN {X 0,Y 608.45,Z 232.315,A -85,B 0,C 180,E1 -521.13,E2 -521.13} C_VEL
LIN {X 0,Y 608.454,Z 232.318,A -85,B 0,C 180,E1 -523.905,E2 -523.905} C_VEL
LIN {X 0,Y 608.466,Z 232.311,A -85,B 0,C 180,E1 -526.643,E2 -526.643} C_VEL
LIN {X 0,Y 608.466,Z 232.318,A -85,B 0,C 180,E1 -529.349,E2 -529.349} C_VEL
LIN {X 0,Y 608.464,Z 232.313,A -85,B 0,C 180,E1 -532.032,E2 -532.032} C_VEL
LIN {X 0,Y 608.467,Z 232.312,A -85,B 0,C 180,E1 -534.697,E2 -534.697} C_VEL
LIN {X 0,Y 608.479,Z 232.32,A -85,B 0,C 180,E1 -537.351,E2 -537.351} C_VEL
LIN {X 0,Y 608.459,Z 232.312,A -85,B 0,C 180,E1 -539.999,E2 -539.999} C_VEL
LIN {X 0,Y 608.481,Z 232.311,A -85,B 0,C 180,E1 -542.647,E2 -542.647} C_VEL
LIN {X 0,Y 608.464,Z 232.319,A -85,B 0,C 180,E1 -545.301,E2 -545.301} C_VEL
LIN {X 0,Y 608.46,Z 232.312,A -85,B 0,C 180,E1 -547.966,E2 -547.966} C_VEL
LIN {X 0,Y 608.451,Z 232.317,A -85,B 0,C 180,E1 -549.472,E2 -549.472} C_VEL
LIN {X 0,Y 607.766,Z 232.4,A -85,B 0,C 180,E1 -550.025,E2 -550.025} C_VEL
LIN {X 0,Y 604.906,Z 232.763,A -85,B 0,C 180,E1 -550.922,E2 -550.922} C_VEL
LIN {X 0,Y 602.506,Z 233.057,A -85,B 0,C 180,E1 -551.643,E2 -551.643} C_VEL
LIN {X 0,Y 601.482,Z 233.182,A -85,B 0,C 180,E1 -552.2,E2 -552.2} C_VEL
LIN {X 0,Y 601.401,Z 233.192,A -85,B 0,C 180,E1 -552.388,E2 -552.388} C_VEL
LIN {X 0,Y 601.423,Z 233.198,A -85,B 0,C 180,E1 -554.896,E2 -554.896} C_VEL
LIN {X 0,Y 601.422,Z 233.198,A -85,B 0,C 180,E1 -556.985,E2 -556.985} C_VEL
LIN {X 0,Y 601.397,Z 233.191,A -85,B 0,C 180,E1 -559.808,E2 -559.808} C_VEL
LIN {X 0,Y 601.442,Z 233.195,A -85,B 0,C 180,E1 -562.681,E2 -562.681} C_VEL
LIN {X 0,Y 601.39,Z 233.2,A -85,B 0,C 180,E1 -564.878,E2 -564.878} C_VEL
LIN {X 0,Y 601.412,Z 233.19,A -85,B 0,C 180,E1 -567.866,E2 -567.866} C_VEL
LIN {X 0,Y 601.434,Z 233.19,A -85,B 0,C 180,E1 -570.162,E2 -570.162} C_VEL
LIN {X 0,Y 601.413,Z 233.19,A -85,B 0,C 180,E1 -573.313,E2 -573.313} C_VEL
LIN {X 0,Y 601.431,Z 233.193,A -85,B 0,C 180,E1 -576.266,E2 -576.266} C_VEL
LIN {X 0,Y 601.416,Z 233.19,A -85,B 0,C 180,E1 -579.124,E2 -579.124} C_VEL
LIN {X 0,Y 601.416,Z 233.191,A -85,B 0,C 180,E1 -581.764,E2 -581.764} C_VEL
LIN {X 0,Y 601.407,Z 233.197,A -85,B 0,C 180,E1 -584.535,E2 -584.535} C_VEL
LIN {X 0,Y 601.402,Z 233.191,A -85,B 0,C 180,E1 -587.408,E2 -587.408} C_VEL
LIN {X 0,Y 601.426,Z 233.194,A -85,B 0,C 180,E1 -590.464,E2 -590.464} C_VEL
LIN {X 0,Y 601.416,Z 233.193,A -85,B 0,C 180,E1 -592.618,E2 -592.618} C_VEL
LIN {X 0,Y 601.403,Z 233.223,A -85,B 0,C 180,E1 -595.17,E2 -595.17} C_VEL
LIN {X 0,Y 601.543,Z 242.114,A -85,B 0,C 180,E1 -596.494,E2 -596.494} C_VEL
LIN {X 0,Y 601.519,Z 259.652,A -85,B 0,C 180,E1 -599.065,E2 -599.065} C_VEL
LIN {X 0,Y 601.468,Z 266.895,A -85,B 0,C 180,E1 -600.096,E2 -600.096} C_VEL
LIN {X 0,Y 601.799,Z 270.354,A -85,B 0,C 180,E1 -600.147,E2 -600.147} C_VEL
LIN {X 0,Y 601.727,Z 403.203,A -85,B 0,C 180,E1 -601.77,E2 -601.77} C_VEL
LIN {X 0,Y 601.686,Z 417.777,A -85,B 0,C 180,E1 -602.088,E2 -602.088} C_VEL
LIN {X 0,Y 601.662,Z 430.363,A -85,B 0,C 180,E1 -602.483,E2 -602.483} C_VEL
LIN {X 0,Y 601.62,Z 442.699,A -85,B 0,C 180,E1 -602.992,E2 -602.992} C_VEL
LIN {X 0,Y 601.546,Z 455.189,A -85,B 0,C 180,E1 -603.644,E2 -603.644} C_VEL
LIN {X 0,Y 601.508,Z 466.727,A -85,B 0,C 180,E1 -604.387,E2 -604.387} C_VEL
LIN {X 0,Y 601.468,Z 478.194,A -85,B 0,C 180,E1 -605.287,E2 -605.287} C_VEL
LIN {X 0,Y 601.441,Z 488.095,A -85,B 0,C 180,E1 -606.226,E2 -606.226} C_VEL
LIN {X 0,Y 601.413,Z 497.643,A -85,B 0,C 180,E1 -607.318,E2 -607.318} C_VEL
LIN {X 0,Y 601.394,Z 505.447,A -85,B 0,C 180,E1 -608.401,E2 -608.401} C_VEL
LIN {X 0,Y 601.357,Z 511.819,A -85,B 0,C 180,E1 -609.476,E2 -609.476} C_VEL
LIN {X 0,Y 601.355,Z 516.995,A -85,B 0,C 180,E1 -610.545,E2 -610.545} C_VEL
LIN {X 0,Y 601.325,Z 521.12,A -85,B 0,C 180,E1 -611.606,E2 -611.606} C_VEL
LIN {X 0,Y 601.333,Z 525.076,A -85,B 0,C 180,E1 -613.012,E2 -613.012} C_VEL
LIN {X 0,Y 601.321,Z 527.483,A -85,B 0,C 180,E1 -614.407,E2 -614.407} C_VEL
LIN {X 0,Y 601.329,Z 528.448,A -85,B 0,C 180,E1 -615.793,E2 -615.793} C_VEL
LIN {X 0,Y 601.319,Z 528.016,A -85,B 0,C 180,E1 -617.17,E2 -617.17} C_VEL
LIN {X 0,Y 601.315,Z 526.2,A -85,B 0,C 180,E1 -618.54,E2 -618.54} C_VEL
LIN {X 0,Y 601.33,Z 522.953,A -85,B 0,C 180,E1 -619.904,E2 -619.904} C_VEL
LIN {X 0,Y 601.344,Z 518.196,A -85,B 0,C 180,E1 -621.261,E2 -621.261} C_VEL
LIN {X 0,Y 601.372,Z 513.596,A -85,B 0,C 180,E1 -622.277,E2 -622.277} C_VEL
LIN {X 0,Y 601.384,Z 507.477,A -85,B 0,C 180,E1 -623.37,E2 -623.37} C_VEL
LIN {X 0,Y 601.408,Z 499.999,A -85,B 0,C 180,E1 -624.468,E2 -624.468} C_VEL
LIN {X 0,Y 601.432,Z 491.714,A -85,B 0,C 180,E1 -625.476,E2 -625.476} C_VEL
LIN {X 0,Y 601.471,Z 481.799,A -85,B 0,C 180,E1 -626.483,E2 -626.483} C_VEL
LIN {X 0,Y 601.5,Z 470.788,A -85,B 0,C 180,E1 -627.405,E2 -627.405} C_VEL
LIN {X 0,Y 601.562,Z 458.545,A -85,B 0,C 180,E1 -628.243,E2 -628.243} C_VEL
LIN {X 0,Y 601.592,Z 446.508,A -85,B 0,C 180,E1 -628.912,E2 -628.912} C_VEL
LIN {X 0,Y 601.645,Z 433.212,A -85,B 0,C 180,E1 -629.498,E2 -629.498} C_VEL
LIN {X 0,Y 601.685,Z 419.339,A -85,B 0,C 180,E1 -629.958,E2 -629.958} C_VEL
LIN {X 0,Y 601.693,Z 405.821,A -85,B 0,C 180,E1 -630.272,E2 -630.272} C_VEL
LIN {X 0,Y 601.706,Z 384.308,A -85,B 0,C 180,E1 -630.565,E2 -630.565} C_VEL
LIN {X 0,Y 601.675,Z 268.166,A -85,B 0,C 180,E1 -631.973,E2 -631.973} C_VEL
LIN {X 0,Y 601.448,Z 266.667,A -85,B 0,C 180,E1 -632.009,E2 -632.009} C_VEL
LIN {X 0,Y 601.577,Z 247.107,A -85,B 0,C 180,E1 -634.859,E2 -634.859} C_VEL
LIN {X 0,Y 601.453,Z 233.288,A -85,B 0,C 180,E1 -636.908,E2 -636.908} C_VEL
LIN {X 0,Y 601.41,Z 233.193,A -85,B 0,C 180,E1 -639.416,E2 -639.416} C_VEL
LIN {X 0,Y 601.415,Z 233.196,A -85,B 0,C 180,E1 -642.142,E2 -642.142} C_VEL
LIN {X 0,Y 601.421,Z 233.189,A -85,B 0,C 180,E1 -644.897,E2 -644.897} C_VEL
LIN {X 0,Y 601.424,Z 233.188,A -85,B 0,C 180,E1 -646.986,E2 -646.986} C_VEL
LIN {X 0,Y 601.399,Z 233.201,A -85,B 0,C 180,E1 -649.809,E2 -649.809} C_VEL
LIN {X 0,Y 601.406,Z 233.19,A -85,B 0,C 180,E1 -652.683,E2 -652.683} C_VEL
LIN {X 0,Y 601.396,Z 233.192,A -85,B 0,C 180,E1 -654.878,E2 -654.878} C_VEL
LIN {X 0,Y 601.416,Z 233.195,A -85,B 0,C 180,E1 -657.867,E2 -657.867} C_VEL
LIN {X 0,Y 601.434,Z 233.189,A -85,B 0,C 180,E1 -660.163,E2 -660.163} C_VEL
LIN {X 0,Y 601.421,Z 233.189,A -85,B 0,C 180,E1 -662.718,E2 -662.718} C_VEL
LIN {X 0,Y 601.405,Z 233.195,A -85,B 0,C 180,E1 -665.116,E2 -665.116} C_VEL
LIN {X 0,Y 601.423,Z 233.198,A -85,B 0,C 180,E1 -667.419,E2 -667.419} C_VEL
LIN {X 0,Y 601.404,Z 233.192,A -85,B 0,C 180,E1 -669.995,E2 -669.995} C_VEL
LIN {X 0,Y 601.427,Z 233.189,A -85,B 0,C 180,E1 -672.668,E2 -672.668} C_VEL
LIN {X 0,Y 601.41,Z 233.197,A -85,B 0,C 180,E1 -675.483,E2 -675.483} C_VEL
LIN {X 0,Y 601.416,Z 233.189,A -85,B 0,C 180,E1 -678.406,E2 -678.406} C_VEL
LIN {X 0,Y 601.429,Z 233.192,A -85,B 0,C 180,E1 -680.877,E2 -680.877} C_VEL
LIN {X 0,Y 601.434,Z 233.189,A -85,B 0,C 180,E1 -683.734,E2 -683.734} C_VEL
LIN {X 0,Y 601.425,Z 233.188,A -85,B 0,C 180,E1 -686.064,E2 -686.064} C_VEL
LIN {X 0,Y 601.43,Z 233.19,A -85,B 0,C 180,E1 -688.542,E2 -688.542} C_VEL
LIN {X 0,Y 601.426,Z 233.192,A -85,B 0,C 180,E1 -691.374,E2 -691.374} C_VEL
LIN {X 0,Y 601.398,Z 233.192,A -85,B 0,C 180,E1 -693.637,E2 -693.637} C_VEL
LIN {X 0,Y 601.415,Z 233.194,A -85,B 0,C 180,E1 -696.591,E2 -696.591} C_VEL
LIN {X 0,Y 601.424,Z 233.19,A -85,B 0,C 180,E1 -699.479,E2 -699.479} C_VEL
LIN {X 0,Y 601.395,Z 233.194,A -85,B 0,C 180,E1 -702.313,E2 -702.313} C_VEL
LIN {X 0,Y 601.412,Z 233.194,A -85,B 0,C 180,E1 -704.41,E2 -704.41} C_VEL
LIN {X 0,Y 601.421,Z 233.192,A -85,B 0,C 180,E1 -707.173,E2 -707.173} C_VEL
LIN {X 0,Y 601.427,Z 233.188,A -85,B 0,C 180,E1 -709.906,E2 -709.906} C_VEL
LIN {X 0,Y 601.446,Z 233.196,A -85,B 0,C 180,E1 -712.616,E2 -712.616} C_VEL
LIN {X 0,Y 601.422,Z 233.189,A -85,B 0,C 180,E1 -715.309,E2 -715.309} C_VEL
LIN {X 0,Y 601.418,Z 233.191,A -85,B 0,C 180,E1 -717.992,E2 -717.992} C_VEL
LIN {X 0,Y 601.447,Z 233.192,A -85,B 0,C 180,E1 -720.67,E2 -720.67} C_VEL
LIN {X 0,Y 601.427,Z 233.188,A -85,B 0,C 180,E1 -723.35,E2 -723.35} C_VEL
LIN {X 0,Y 601.406,Z 233.195,A -85,B 0,C 180,E1 -726.038,E2 -726.038} C_VEL
LIN {X 0,Y 601.433,Z 233.191,A -85,B 0,C 180,E1 -728.738,E2 -728.738} C_VEL
LIN {X 0,Y 601.429,Z 233.188,A -85,B 0,C 180,E1 -731.459,E2 -731.459} C_VEL
LIN {X 0,Y 601.412,Z 233.2,A -85,B 0,C 180,E1 -734.206,E2 -734.206} C_VEL
LIN {X 0,Y 601.428,Z 233.188,A -85,B 0,C 180,E1 -736.987,E2 -736.987} C_VEL
LIN {X 0,Y 601.407,Z 233.195,A -85,B 0,C 180,E1 -739.81,E2 -739.81} C_VEL
LIN {X 0,Y 601.406,Z 233.192,A -85,B 0,C 180,E1 -742.684,E2 -742.684} C_VEL
LIN {X 0,Y 601.401,Z 233.191,A -85,B 0,C 180,E1 -744.879,E2 -744.879} C_VEL
LIN {X 0,Y 601.417,Z 233.197,A -85,B 0,C 180,E1 -747.868,E2 -747.868} C_VEL
LIN {X 0,Y 601.444,Z 233.192,A -85,B 0,C 180,E1 -750.164,E2 -750.164} C_VEL
LIN {X 0,Y 601.413,Z 233.19,A -85,B 0,C 180,E1 -752.716,E2 -752.716} C_VEL
LIN {X 0,Y 601.411,Z 233.19,A -85,B 0,C 180,E1 -755.116,E2 -755.116} C_VEL
LIN {X 0,Y 601.432,Z 233.191,A -85,B 0,C 180,E1 -757.42,E2 -757.42} C_VEL
LIN {X 0,Y 601.409,Z 233.196,A -85,B 0,C 180,E1 -759.996,E2 -759.996} C_VEL
LIN {X 0,Y 601.407,Z 233.19,A -85,B 0,C 180,E1 -762.671,E2 -762.671} C_VEL
LIN {X 0,Y 601.424,Z 233.195,A -85,B 0,C 180,E1 -765.483,E2 -765.483} C_VEL
LIN {X 0,Y 601.423,Z 233.189,A -85,B 0,C 180,E1 -768.408,E2 -768.408} C_VEL
LIN {X 0,Y 601.428,Z 233.198,A -85,B 0,C 180,E1 -771.53,E2 -771.53} C_VEL
LIN {X 0,Y 601.385,Z 233.193,A -85,B 0,C 180,E1 -774.246,E2 -774.246} C_VEL
LIN {X 0,Y 601.427,Z 233.188,A -85,B 0,C 180,E1 -776.687,E2 -776.687} C_VEL
LIN {X 0,Y 601.412,Z 233.195,A -85,B 0,C 180,E1 -779.058,E2 -779.058} C_VEL
LIN {X 0,Y 601.432,Z 233.198,A -85,B 0,C 180,E1 -781.374,E2 -781.374} C_VEL
LIN {X 0,Y 601.4,Z 233.197,A -85,B 0,C 180,E1 -783.637,E2 -783.637} C_VEL
LIN {X 0,Y 601.437,Z 233.314,A -85,B 0,C 180,E1 -786.18,E2 -786.18} C_VEL
LIN {X 0,Y 601.752,Z 236.493,A -85,B 0,C 180,E1 -786.604,E2 -786.604} C_VEL
LIN {X 0,Y 601.661,Z 259.102,A -85,B 0,C 180,E1 -789.487,E2 -789.487} C_VEL
LIN {X 0,Y 601.583,Z 281.71,A -85,B 0,C 180,E1 -792.318,E2 -792.318} C_VEL
LIN {X 0,Y 601.539,Z 295.62,A -85,B 0,C 180,E1 -794.037,E2 -794.037} C_VEL
LIN {X 0,Y 601.835,Z 299.638,A -85,B 0,C 180,E1 -794.094,E2 -794.094} C_VEL
LIN {X 0,Y 601.716,Z 433.994,A -85,B 0,C 180,E1 -795.739,E2 -795.739} C_VEL
LIN {X 0,Y 601.709,Z 448.584,A -85,B 0,C 180,E1 -796.066,E2 -796.066} C_VEL
LIN {X 0,Y 601.664,Z 462.84,A -85,B 0,C 180,E1 -796.533,E2 -796.533} C_VEL
LIN {X 0,Y 601.605,Z 475.638,A -85,B 0,C 180,E1 -797.09,E2 -797.09} C_VEL
LIN {X 0,Y 601.543,Z 488.097,A -85,B 0,C 180,E1 -797.775,E2 -797.775} C_VEL
LIN {X 0,Y 601.504,Z 499.475,A -85,B 0,C 180,E1 -798.543,E2 -798.543} C_VEL
LIN {X 0,Y 601.482,Z 509.934,A -85,B 0,C 180,E1 -799.396,E2 -799.396} C_VEL
LIN {X 0,Y 601.43,Z 520.335,A -85,B 0,C 180,E1 -800.415,E2 -800.415} C_VEL
LIN {X 0,Y 601.407,Z 528.914,A -85,B 0,C 180,E1 -801.431,E2 -801.431} C_VEL
LIN {X 0,Y 601.392,Z 537.114,A -85,B 0,C 180,E1 -802.614,E2 -802.614} C_VEL
LIN {X 0,Y 601.361,Z 542.752,A -85,B 0,C 180,E1 -803.605,E2 -803.605} C_VEL
LIN {X 0,Y 601.355,Z 547.568,A -85,B 0,C 180,E1 -804.635,E2 -804.635} C_VEL
LIN {X 0,Y 601.343,Z 552.442,A -85,B 0,C 180,E1 -805.979,E2 -805.979} C_VEL
LIN {X 0,Y 601.324,Z 555.831,A -85,B 0,C 180,E1 -807.32,E2 -807.32} C_VEL
LIN {X 0,Y 601.342,Z 557.831,A -85,B 0,C 180,E1 -808.661,E2 -808.661} C_VEL
LIN {X 0,Y 601.333,Z 558.5,A -85,B 0,C 180,E1 -810,E2 -810} C_VEL
LIN {X 0,Y 601.342,Z 557.831,A -85,B 0,C 180,E1 -811.339,E2 -811.339} C_VEL
LIN {X 0,Y 601.324,Z 555.832,A -85,B 0,C 180,E1 -812.679,E2 -812.679} C_VEL
LIN {X 0,Y 601.343,Z 552.443,A -85,B 0,C 180,E1 -814.021,E2 -814.021} C_VEL
LIN {X 0,Y 601.355,Z 547.568,A -85,B 0,C 180,E1 -815.365,E2 -815.365} C_VEL
LIN {X 0,Y 601.372,Z 541.624,A -85,B 0,C 180,E1 -816.605,E2 -816.605} C_VEL
LIN {X 0,Y 601.386,Z 534.921,A -85,B 0,C 180,E1 -817.723,E2 -817.723} C_VEL
LIN {X 0,Y 601.412,Z 526.2,A -85,B 0,C 180,E1 -818.907,E2 -818.907} C_VEL
LIN {X 0,Y 601.433,Z 517.084,A -85,B 0,C 180,E1 -819.925,E2 -819.925} C_VEL
LIN {X 0,Y 601.497,Z 506.831,A -85,B 0,C 180,E1 -820.876,E2 -820.876} C_VEL
LIN {X 0,Y 601.533,Z 495.975,A -85,B 0,C 180,E1 -821.712,E2 -821.712} C_VEL
LIN {X 0,Y 601.575,Z 483.783,A -85,B 0,C 180,E1 -822.481,E2 -822.481} C_VEL
LIN {X 0,Y 601.628,Z 470.136,A -85,B 0,C 180,E1 -823.167,E2 -823.167} C_VEL
LIN {X 0,Y 601.681,Z 456.922,A -85,B 0,C 180,E1 -823.679,E2 -823.679} C_VEL
LIN {X 0,Y 601.714,Z 442.693,A -85,B 0,C 180,E1 -824.083,E2 -824.083} C_VEL
LIN {X 0,Y 601.71,Z 429.215,A -85,B 0,C 180,E1 -824.334,E2 -824.334} C_VEL
LIN {X 0,Y 601.742,Z 296.868,A -85,B 0,C 180,E1 -825.942,E2 -825.942} C_VEL
LIN {X 0,Y 601.539,Z 295.489,A -85,B 0,C 180,E1 -825.979,E2 -825.979} C_VEL
LIN {X 0,Y 601.598,Z 274.149,A -85,B 0,C 180,E1 -828.624,E2 -828.624} C_VEL
LIN {X 0,Y 601.658,Z 252.038,A -85,B 0,C 180,E1 -831.409,E2 -831.409} C_VEL
LIN {X 0,Y 601.766,Z 235.081,A -85,B 0,C 180,E1 -833.578,E2 -833.578} C_VEL
LIN {X 0,Y 601.414,Z 233.194,A -85,B 0,C 180,E1 -833.867,E2 -833.867} C_VEL
LIN {X 0,Y 601.399,Z 233.198,A -85,B 0,C 180,E1 -836.363,E2 -836.363} C_VEL
LIN {X 0,Y 601.439,Z 233.194,A -85,B 0,C 180,E1 -838.789,E2 -838.789} C_VEL
LIN {X 0,Y 601.406,Z 233.191,A -85,B 0,C 180,E1 -841.726,E2 -841.726} C_VEL
LIN {X 0,Y 601.428,Z 233.192,A -85,B 0,C 180,E1 -844.117,E2 -844.117} C_VEL
LIN {X 0,Y 601.433,Z 233.187,A -85,B 0,C 180,E1 -847.381,E2 -847.381} C_VEL
LIN {X 0,Y 601.399,Z 233.196,A -85,B 0,C 180,E1 -849.995,E2 -849.995} C_VEL
LIN {X 0,Y 601.413,Z 233.194,A -85,B 0,C 180,E1 -852.669,E2 -852.669} C_VEL
LIN {X 0,Y 601.422,Z 233.189,A -85,B 0,C 180,E1 -855.481,E2 -855.481} C_VEL
LIN {X 0,Y 601.42,Z 233.195,A -85,B 0,C 180,E1 -858.406,E2 -858.406} C_VEL
LIN {X 0,Y 601.434,Z 233.188,A -85,B 0,C 180,E1 -860.875,E2 -860.875} C_VEL
LIN {X 0,Y 601.44,Z 233.191,A -85,B 0,C 180,E1 -863.733,E2 -863.733} C_VEL
LIN {X 0,Y 601.428,Z 233.198,A -85,B 0,C 180,E1 -866.063,E2 -866.063} C_VEL
LIN {X 0,Y 601.435,Z 233.188,A -85,B 0,C 180,E1 -868.541,E2 -868.541} C_VEL
LIN {X 0,Y 601.427,Z 233.19,A -85,B 0,C 180,E1 -871.372,E2 -871.372} C_VEL
LIN {X 0,Y 601.4,Z 233.198,A -85,B 0,C 180,E1 -873.636,E2 -873.636} C_VEL
LIN {X 0,Y 601.414,Z 233.19,A -85,B 0,C 180,E1 -876.589,E2 -876.589} C_VEL
LIN {X 0,Y 601.427,Z 233.194,A -85,B 0,C 180,E1 -879.477,E2 -879.477} C_VEL
LIN {X 0,Y 601.393,Z 233.193,A -85,B 0,C 180,E1 -882.311,E2 -882.311} C_VEL
LIN {X 0,Y 601.412,Z 233.19,A -85,B 0,C 180,E1 -884.408,E2 -884.408} C_VEL
LIN {X 0,Y 601.422,Z 233.192,A -85,B 0,C 180,E1 -887.171,E2 -887.171} C_VEL
LIN {X 0,Y 601.424,Z 233.192,A -85,B 0,C 180,E1 -889.904,E2 -889.904} C_VEL
LIN {X 0,Y 601.446,Z 233.185,A -85,B 0,C 180,E1 -892.614,E2 -892.614} C_VEL
LIN {X 0,Y 601.431,Z 233.197,A -85,B 0,C 180,E1 -895.307,E2 -895.307} C_VEL
LIN {X 0,Y 601.41,Z 233.191,A -85,B 0,C 180,E1 -897.99,E2 -897.99} C_VEL
LIN {X 0,Y 601.449,Z 233.187,A -85,B 0,C 180,E1 -900.669,E2 -900.669} C_VEL
LIN {X 0,Y 601.429,Z 233.196,A -85,B 0,C 180,E1 -903.349,E2 -903.349} C_VEL
LIN {X 0,Y 601.397,Z 233.191,A -85,B 0,C 180,E1 -906.036,E2 -906.036} C_VEL
LIN {X 0,Y 601.433,Z 233.191,A -85,B 0,C 180,E1 -908.737,E2 -908.737} C_VEL
LIN {X 0,Y 601.425,Z 233.192,A -85,B 0,C 180,E1 -911.457,E2 -911.457} C_VEL
LIN {X 0,Y 601.401,Z 233.192,A -85,B 0,C 180,E1 -912.388,E2 -912.388} C_VEL
LIN {X 0,Y 600.742,Z 233.283,A -85,B 0,C 180,E1 -912.948,E2 -912.948} C_VEL
LIN {X 0,Y 597.892,Z 233.64,A -85,B 0,C 180,E1 -913.855,E2 -913.855} C_VEL
LIN {X 0,Y 595.477,Z 233.94,A -85,B 0,C 180,E1 -914.586,E2 -914.586} C_VEL
LIN {X 0,Y 594.438,Z 234.066,A -85,B 0,C 180,E1 -915.149,E2 -915.149} C_VEL
LIN {X 0,Y 594.352,Z 234.073,A -85,B 0,C 180,E1 -915.34,E2 -915.34} C_VEL
LIN {X 0,Y 594.378,Z 234.071,A -85,B 0,C 180,E1 -917.193,E2 -917.193} C_VEL
LIN {X 0,Y 594.368,Z 234.067,A -85,B 0,C 180,E1 -920.053,E2 -920.053} C_VEL
LIN {X 0,Y 594.386,Z 234.072,A -85,B 0,C 180,E1 -922.965,E2 -922.965} C_VEL
LIN {X 0,Y 594.36,Z 234.071,A -85,B 0,C 180,E1 -925.192,E2 -925.192} C_VEL
LIN {X 0,Y 594.37,Z 234.067,A -85,B 0,C 180,E1 -927.526,E2 -927.526} C_VEL
LIN {X 0,Y 594.384,Z 234.07,A -85,B 0,C 180,E1 -930.33,E2 -930.33} C_VEL
LIN {X 0,Y 594.365,Z 234.072,A -85,B 0,C 180,E1 -932.949,E2 -932.949} C_VEL
LIN {X 0,Y 594.342,Z 234.07,A -85,B 0,C 180,E1 -935.408,E2 -935.408} C_VEL
LIN {X 0,Y 594.377,Z 234.069,A -85,B 0,C 180,E1 -937.94,E2 -937.94} C_VEL
LIN {X 0,Y 594.368,Z 234.071,A -85,B 0,C 180,E1 -940.822,E2 -940.822} C_VEL
LIN {X 0,Y 594.369,Z 234.067,A -85,B 0,C 180,E1 -943.297,E2 -943.297} C_VEL
LIN {X 0,Y 594.366,Z 234.076,A -85,B 0,C 180,E1 -946.159,E2 -946.159} C_VEL
LIN {X 0,Y 594.367,Z 234.068,A -85,B 0,C 180,E1 -949.177,E2 -949.177} C_VEL
LIN {X 0,Y 594.376,Z 234.076,A -85,B 0,C 180,E1 -952.06,E2 -952.06} C_VEL
LIN {X 0,Y 594.338,Z 234.077,A -85,B 0,C 180,E1 -954.676,E2 -954.676} C_VEL
LIN {X 0,Y 594.379,Z 234.206,A -85,B 0,C 180,E1 -955.06,E2 -955.06} C_VEL
LIN {X 0,Y 594.611,Z 239.24,A -85,B 0,C 180,E1 -955.826,E2 -955.826} C_VEL
LIN {X 0,Y 594.49,Z 257.221,A -85,B 0,C 180,E1 -958.499,E2 -958.499} C_VEL
LIN {X 0,Y 594.463,Z 266.722,A -85,B 0,C 180,E1 -959.896,E2 -959.896} C_VEL
LIN {X 0,Y 594.99,Z 271.352,A -85,B 0,C 180,E1 -959.973,E2 -959.973} C_VEL
LIN {X 0,Y 594.861,Z 403.493,A -85,B 0,C 180,E1 -961.607,E2 -961.607} C_VEL
LIN {X 0,Y 594.788,Z 417.975,A -85,B 0,C 180,E1 -961.928,E2 -961.928} C_VEL
LIN {X 0,Y 594.742,Z 431.514,A -85,B 0,C 180,E1 -962.367,E2 -962.367} C_VEL
LIN {X 0,Y 594.666,Z 444.703,A -85,B 0,C 180,E1 -962.935,E2 -962.935} C_VEL
LIN {X 0,Y 594.585,Z 457.985,A -85,B 0,C 180,E1 -963.667,E2 -963.667} C_VEL
LIN {X 0,Y 594.504,Z 469.302,A -85,B 0,C 180,E1 -964.439,E2 -964.439} C_VEL
LIN {X 0,Y 594.46,Z 480.796,A -85,B 0,C 180,E1 -965.39,E2 -965.39} C_VEL
LIN {X 0,Y 594.408,Z 489.881,A -85,B 0,C 180,E1 -966.297,E2 -966.297} C_VEL
LIN {X 0,Y 594.344,Z 498.059,A -85,B 0,C 180,E1 -967.265,E2 -967.265} C_VEL
LIN {X 0,Y 594.336,Z 505.475,A -85,B 0,C 180,E1 -968.314,E2 -968.314} C_VEL
LIN {X 0,Y 594.284,Z 512.802,A -85,B 0,C 180,E1 -969.583,E2 -969.583} C_VEL
LIN {X 0,Y 594.274,Z 517.763,A -85,B 0,C 180,E1 -970.663,E2 -970.663} C_VEL
LIN {X 0,Y 594.245,Z 521.695,A -85,B 0,C 180,E1 -971.736,E2 -971.736} C_VEL
LIN {X 0,Y 594.239,Z 524.698,A -85,B 0,C 180,E1 -972.803,E2 -972.803} C_VEL
LIN {X 0,Y 594.247,Z 527.285,A -85,B 0,C 180,E1 -974.216,E2 -974.216} C_VEL
LIN {X 0,Y 594.237,Z 528.409,A -85,B 0,C 180,E1 -975.62,E2 -975.62} C_VEL
LIN {X 0,Y 594.236,Z 528.132,A -85,B 0,C 180,E1 -977.014,E2 -977.014} C_VEL
LIN {X 0,Y 594.227,Z 526.476,A -85,B 0,C 180,E1 -978.401,E2 -978.401} C_VEL
LIN {X 0,Y 594.229,Z 523.411,A -85,B 0,C 180,E1 -979.782,E2 -979.782} C_VEL
LIN {X 0,Y 594.267,Z 518.877,A -85,B 0,C 180,E1 -981.156,E2 -981.156} C_VEL
LIN {X 0,Y 594.288,Z 514.389,A -85,B 0,C 180,E1 -982.184,E2 -982.184} C_VEL
LIN {X 0,Y 594.33,Z 508.103,A -85,B 0,C 180,E1 -983.352,E2 -983.352} C_VEL
LIN {X 0,Y 594.327,Z 499.978,A -85,B 0,C 180,E1 -984.572,E2 -984.572} C_VEL
LIN {X 0,Y 594.379,Z 491.687,A -85,B 0,C 180,E1 -985.592,E2 -985.592} C_VEL
LIN {X 0,Y 594.441,Z 481.766,A -85,B 0,C 180,E1 -986.611,E2 -986.611} C_VEL
LIN {X 0,Y 594.499,Z 470.746,A -85,B 0,C 180,E1 -987.544,E2 -987.544} C_VEL
LIN {X 0,Y 594.6,Z 458.486,A -85,B 0,C 180,E1 -988.392,E2 -988.392} C_VEL
LIN {X 0,Y 594.643,Z 446.438,A -85,B 0,C 180,E1 -989.069,E2 -989.069} C_VEL
LIN {X 0,Y 594.722,Z 433.116,A -85,B 0,C 180,E1 -989.662,E2 -989.662} C_VEL
LIN {X 0,Y 594.783,Z 419.2,A -85,B 0,C 180,E1 -990.127,E2 -990.127} C_VEL
LIN {X 0,Y 594.822,Z 405.583,A -85,B 0,C 180,E1 -990.444,E2 -990.444} C_VEL
LIN {X 0,Y 594.859,Z 382.179,A -85,B 0,C 180,E1 -990.762,E2 -990.762} C_VEL
LIN {X 0,Y 594.883,Z 269.149,A -85,B 0,C 180,E1 -992.148,E2 -992.148} C_VEL
LIN {X 0,Y 594.468,Z 266.664,A -85,B 0,C 180,E1 -992.202,E2 -992.202} C_VEL
LIN {X 0,Y 594.625,Z 247.117,A -85,B 0,C 180,E1 -995.086,E2 -995.086} C_VEL
LIN {X 0,Y 594.595,Z 235.259,A -85,B 0,C 180,E1 -996.863,E2 -996.863} C_VEL
LIN {X 0,Y 594.391,Z 234.069,A -85,B 0,C 180,E1 -997.084,E2 -997.084} C_VEL
LIN {X 0,Y 594.364,Z 234.072,A -85,B 0,C 180,E1 -999.529,E2 -999.529} C_VEL
LIN {X 0,Y 594.386,Z 234.069,A -85,B 0,C 180,E1 -1002.288,E2 -1002.288} C_VEL
LIN {X 0,Y 594.365,Z 234.069,A -85,B 0,C 180,E1 -1005.078,E2 -1005.078} C_VEL
LIN {X 0,Y 594.381,Z 234.067,A -85,B 0,C 180,E1 -1007.193,E2 -1007.193} C_VEL
LIN {X 0,Y 594.369,Z 234.072,A -85,B 0,C 180,E1 -1010.054,E2 -1010.054} C_VEL
LIN {X 0,Y 594.356,Z 234.069,A -85,B 0,C 180,E1 -1012.967,E2 -1012.967} C_VEL
LIN {X 0,Y 594.371,Z 234.069,A -85,B 0,C 180,E1 -1015.193,E2 -1015.193} C_VEL
LIN {X 0,Y 594.37,Z 234.075,A -85,B 0,C 180,E1 -1017.527,E2 -1017.527} C_VEL
LIN {X 0,Y 594.387,Z 234.065,A -85,B 0,C 180,E1 -1020.331,E2 -1020.331} C_VEL
LIN {X 0,Y 594.371,Z 234.068,A -85,B 0,C 180,E1 -1022.95,E2 -1022.95} C_VEL
LIN {X 0,Y 594.371,Z 234.076,A -85,B 0,C 180,E1 -1025.407,E2 -1025.407} C_VEL
LIN {X 0,Y 594.377,Z 234.069,A -85,B 0,C 180,E1 -1027.94,E2 -1027.94} C_VEL
LIN {X 0,Y 594.379,Z 234.068,A -85,B 0,C 180,E1 -1030.824,E2 -1030.824} C_VEL
LIN {X 0,Y 594.373,Z 234.076,A -85,B 0,C 180,E1 -1033.298,E2 -1033.298} C_VEL
LIN {X 0,Y 594.367,Z 234.067,A -85,B 0,C 180,E1 -1036.159,E2 -1036.159} C_VEL
LIN {X 0,Y 594.373,Z 234.067,A -85,B 0,C 180,E1 -1038.537,E2 -1038.537} C_VEL
LIN {X 0,Y 594.379,Z 234.074,A -85,B 0,C 180,E1 -1041.295,E2 -1041.295} C_VEL
LIN {X 0,Y 594.386,Z 234.066,A -85,B 0,C 180,E1 -1043.76,E2 -1043.76} C_VEL
LIN {X 0,Y 594.371,Z 234.067,A -85,B 0,C 180,E1 -1046.24,E2 -1046.24} C_VEL
LIN {X 0,Y 594.38,Z 234.069,A -85,B 0,C 180,E1 -1048.652,E2 -1048.652} C_VEL
LIN {X 0,Y 594.375,Z 234.076,A -85,B 0,C 180,E1 -1051.041,E2 -1051.041} C_VEL
LIN {X 0,Y 594.381,Z 234.07,A -85,B 0,C 180,E1 -1053.302,E2 -1053.302} C_VEL
LIN {X 0,Y 594.387,Z 234.066,A -85,B 0,C 180,E1 -1056.297,E2 -1056.297} C_VEL
LIN {X 0,Y 594.394,Z 234.068,A -85,B 0,C 180,E1 -1059.225,E2 -1059.225} C_VEL
LIN {X 0,Y 594.374,Z 234.067,A -85,B 0,C 180,E1 -1062.097,E2 -1062.097} C_VEL
LIN {X 0,Y 594.365,Z 234.069,A -85,B 0,C 180,E1 -1064.22,E2 -1064.22} C_VEL
LIN {X 0,Y 594.368,Z 234.072,A -85,B 0,C 180,E1 -1067.018,E2 -1067.018} C_VEL
LIN {X 0,Y 594.387,Z 234.065,A -85,B 0,C 180,E1 -1069.785,E2 -1069.785} C_VEL
LIN {X 0,Y 594.394,Z 234.073,A -85,B 0,C 180,E1 -1072.528,E2 -1072.528} C_VEL
LIN {X 0,Y 594.391,Z 234.065,A -85,B 0,C 180,E1 -1075.253,E2 -1075.253} C_VEL
LIN {X 0,Y 594.389,Z 234.066,A -85,B 0,C 180,E1 -1077.968,E2 -1077.968} C_VEL
LIN {X 0,Y 594.418,Z 234.068,A -85,B 0,C 180,E1 -1080.678,E2 -1080.678} C_VEL
LIN {X 0,Y 594.378,Z 234.066,A -85,B 0,C 180,E1 -1083.39,E2 -1083.39} C_VEL
LIN {X 0,Y 594.362,Z 234.073,A -85,B 0,C 180,E1 -1086.11,E2 -1086.11} C_VEL
LIN {X 0,Y 594.394,Z 234.066,A -85,B 0,C 180,E1 -1088.843,E2 -1088.843} C_VEL
LIN {X 0,Y 594.387,Z 234.066,A -85,B 0,C 180,E1 -1091.597,E2 -1091.597} C_VEL
LIN {X 0,Y 594.383,Z 234.073,A -85,B 0,C 180,E1 -1094.378,E2 -1094.378} C_VEL
LIN {X 0,Y 594.387,Z 234.065,A -85,B 0,C 180,E1 -1097.194,E2 -1097.194} C_VEL
LIN {X 0,Y 594.373,Z 234.076,A -85,B 0,C 180,E1 -1100.054,E2 -1100.054} C_VEL
LIN {X 0,Y 594.359,Z 234.068,A -85,B 0,C 180,E1 -1102.968,E2 -1102.968} C_VEL
LIN {X 0,Y 594.372,Z 234.067,A -85,B 0,C 180,E1 -1105.194,E2 -1105.194} C_VEL
LIN {X 0,Y 594.38,Z 234.069,A -85,B 0,C 180,E1 -1107.528,E2 -1107.528} C_VEL
LIN {X 0,Y 594.396,Z 234.067,A -85,B 0,C 180,E1 -1110.332,E2 -1110.332} C_VEL
LIN {X 0,Y 594.373,Z 234.066,A -85,B 0,C 180,E1 -1112.951,E2 -1112.951} C_VEL
LIN {X 0,Y 594.38,Z 234.069,A -85,B 0,C 180,E1 -1115.408,E2 -1115.408} C_VEL
LIN {X 0,Y 594.383,Z 234.073,A -85,B 0,C 180,E1 -1117.941,E2 -1117.941} C_VEL
LIN {X 0,Y 594.374,Z 234.066,A -85,B 0,C 180,E1 -1120.823,E2 -1120.823} C_VEL
LIN {X 0,Y 594.365,Z 234.075,A -85,B 0,C 180,E1 -1123.84,E2 -1123.84} C_VEL
LIN {X 0,Y 594.379,Z 234.066,A -85,B 0,C 180,E1 -1126.703,E2 -1126.703} C_VEL
LIN {X 0,Y 594.369,Z 234.075,A -85,B 0,C 180,E1 -1129.434,E2 -1129.434} C_VEL
LIN {X 0,Y 594.387,Z 234.065,A -85,B 0,C 180,E1 -1132.392,E2 -1132.392} C_VEL
LIN {X 0,Y 594.381,Z 234.075,A -85,B 0,C 180,E1 -1135.421,E2 -1135.421} C_VEL
LIN {X 0,Y 594.383,Z 234.066,A -85,B 0,C 180,E1 -1138.357,E2 -1138.357} C_VEL
LIN {X 0,Y 594.384,Z 234.071,A -85,B 0,C 180,E1 -1141.043,E2 -1141.043} C_VEL
LIN {X 0,Y 594.386,Z 234.068,A -85,B 0,C 180,E1 -1143.978,E2 -1143.978} C_VEL
LIN {X 0,Y 594.421,Z 234.197,A -85,B 0,C 180,E1 -1145.997,E2 -1145.997} C_VEL
LIN {X 0,Y 594.877,Z 237.906,A -85,B 0,C 180,E1 -1146.502,E2 -1146.502} C_VEL
LIN {X 0,Y 594.756,Z 260.515,A -85,B 0,C 180,E1 -1149.419,E2 -1149.419} C_VEL
LIN {X 0,Y 594.598,Z 284.536,A -85,B 0,C 180,E1 -1152.458,E2 -1152.458} C_VEL
LIN {X 0,Y 594.522,Z 295.487,A -85,B 0,C 180,E1 -1153.827,E2 -1153.827} C_VEL
LIN {X 0,Y 595.016,Z 299.638,A -85,B 0,C 180,E1 -1153.907,E2 -1153.907} C_VEL
LIN {X 0,Y 594.856,Z 433.898,A -85,B 0,C 180,E1 -1155.569,E2 -1155.569} C_VEL
LIN {X 0,Y 594.816,Z 448.177,A -85,B 0,C 180,E1 -1155.889,E2 -1155.889} C_VEL
LIN {X 0,Y 594.715,Z 461.72,A -85,B 0,C 180,E1 -1156.329,E2 -1156.329} C_VEL
LIN {X 0,Y 594.65,Z 475.641,A -85,B 0,C 180,E1 -1156.937,E2 -1156.937} C_VEL
LIN {X 0,Y 594.58,Z 488.099,A -85,B 0,C 180,E1 -1157.629,E2 -1157.629} C_VEL
LIN {X 0,Y 594.524,Z 500.562,A -85,B 0,C 180,E1 -1158.488,E2 -1158.488} C_VEL
LIN {X 0,Y 594.449,Z 511.838,A -85,B 0,C 180,E1 -1159.441,E2 -1159.441} C_VEL
LIN {X 0,Y 594.368,Z 521.851,A -85,B 0,C 180,E1 -1160.471,E2 -1160.471} C_VEL
LIN {X 0,Y 594.324,Z 530.171,A -85,B 0,C 180,E1 -1161.5,E2 -1161.5} C_VEL
LIN {X 0,Y 594.303,Z 538.126,A -85,B 0,C 180,E1 -1162.697,E2 -1162.697} C_VEL
LIN {X 0,Y 594.281,Z 544.527,A -85,B 0,C 180,E1 -1163.89,E2 -1163.89} C_VEL
LIN {X 0,Y 594.237,Z 550.199,A -85,B 0,C 180,E1 -1165.251,E2 -1165.251} C_VEL
LIN {X 0,Y 594.259,Z 554.315,A -85,B 0,C 180,E1 -1166.61,E2 -1166.61} C_VEL
LIN {X 0,Y 594.241,Z 557,A -85,B 0,C 180,E1 -1167.967,E2 -1167.967} C_VEL
LIN {X 0,Y 594.237,Z 558.332,A -85,B 0,C 180,E1 -1169.322,E2 -1169.322} C_VEL
LIN {X 0,Y 594.237,Z 558.332,A -85,B 0,C 180,E1 -1170.678,E2 -1170.678} C_VEL
LIN {X 0,Y 594.241,Z 557.001,A -85,B 0,C 180,E1 -1172.033,E2 -1172.033} C_VEL
LIN {X 0,Y 594.259,Z 554.317,A -85,B 0,C 180,E1 -1173.39,E2 -1173.39} C_VEL
LIN {X 0,Y 594.237,Z 550.2,A -85,B 0,C 180,E1 -1174.749,E2 -1174.749} C_VEL
LIN {X 0,Y 594.281,Z 544.528,A -85,B 0,C 180,E1 -1176.11,E2 -1176.11} C_VEL
LIN {X 0,Y 594.303,Z 538.127,A -85,B 0,C 180,E1 -1177.303,E2 -1177.303} C_VEL
LIN {X 0,Y 594.324,Z 530.172,A -85,B 0,C 180,E1 -1178.5,E2 -1178.5} C_VEL
LIN {X 0,Y 594.367,Z 521.853,A -85,B 0,C 180,E1 -1179.528,E2 -1179.528} C_VEL
LIN {X 0,Y 594.449,Z 511.84,A -85,B 0,C 180,E1 -1180.559,E2 -1180.559} C_VEL
LIN {X 0,Y 594.524,Z 500.566,A -85,B 0,C 180,E1 -1181.512,E2 -1181.512} C_VEL
LIN {X 0,Y 594.58,Z 488.102,A -85,B 0,C 180,E1 -1182.371,E2 -1182.371} C_VEL
LIN {X 0,Y 594.65,Z 475.645,A -85,B 0,C 180,E1 -1183.063,E2 -1183.063} C_VEL
LIN {X 0,Y 594.715,Z 461.721,A -85,B 0,C 180,E1 -1183.671,E2 -1183.671} C_VEL
LIN {X 0,Y 594.799,Z 447.57,A -85,B 0,C 180,E1 -1184.128,E2 -1184.128} C_VEL
LIN {X 0,Y 594.858,Z 433.905,A -85,B 0,C 180,E1 -1184.431,E2 -1184.431} C_VEL
LIN {X 0,Y 594.863,Z 297.417,A -85,B 0,C 180,E1 -1186.124,E2 -1186.124} C_VEL
LIN {X 0,Y 594.522,Z 295.489,A -85,B 0,C 180,E1 -1186.173,E2 -1186.173} C_VEL
LIN {X 0,Y 594.65,Z 273.912,A -85,B 0,C 180,E1 -1188.88,E2 -1188.88} C_VEL
LIN {X 0,Y 594.772,Z 253.451,A -85,B 0,C 180,E1 -1191.487,E2 -1191.487} C_VEL
LIN {X 0,Y 594.856,Z 236.494,A -85,B 0,C 180,E1 -1193.684,E2 -1193.684} C_VEL
LIN {X 0,Y 594.391,Z 234.071,A -85,B 0,C 180,E1 -1194.027,E2 -1194.027} C_VEL
LIN {X 0,Y 594.382,Z 234.076,A -85,B 0,C 180,E1 -1196.699,E2 -1196.699} C_VEL
LIN {X 0,Y 594.381,Z 234.07,A -85,B 0,C 180,E1 -1198.998,E2 -1198.998} C_VEL
LIN {X 0,Y 594.383,Z 234.066,A -85,B 0,C 180,E1 -1201.643,E2 -1201.643} C_VEL
LIN {X 0,Y 594.379,Z 234.075,A -85,B 0,C 180,E1 -1204.579,E2 -1204.579} C_VEL
LIN {X 0,Y 594.387,Z 234.065,A -85,B 0,C 180,E1 -1207.608,E2 -1207.608} C_VEL
LIN {X 0,Y 594.368,Z 234.074,A -85,B 0,C 180,E1 -1210.566,E2 -1210.566} C_VEL
LIN {X 0,Y 594.378,Z 234.066,A -85,B 0,C 180,E1 -1213.297,E2 -1213.297} C_VEL
LIN {X 0,Y 594.364,Z 234.077,A -85,B 0,C 180,E1 -1216.159,E2 -1216.159} C_VEL
LIN {X 0,Y 594.377,Z 234.071,A -85,B 0,C 180,E1 -1218.535,E2 -1218.535} C_VEL
LIN {X 0,Y 594.385,Z 234.065,A -85,B 0,C 180,E1 -1221.294,E2 -1221.294} C_VEL
LIN {X 0,Y 594.392,Z 234.069,A -85,B 0,C 180,E1 -1223.758,E2 -1223.758} C_VEL
LIN {X 0,Y 594.374,Z 234.073,A -85,B 0,C 180,E1 -1226.238,E2 -1226.238} C_VEL
LIN {X 0,Y 594.385,Z 234.066,A -85,B 0,C 180,E1 -1228.65,E2 -1228.65} C_VEL
LIN {X 0,Y 594.377,Z 234.066,A -85,B 0,C 180,E1 -1231.041,E2 -1231.041} C_VEL
LIN {X 0,Y 594.384,Z 234.067,A -85,B 0,C 180,E1 -1233.3,E2 -1233.3} C_VEL
LIN {X 0,Y 594.386,Z 234.067,A -85,B 0,C 180,E1 -1236.295,E2 -1236.295} C_VEL
LIN {X 0,Y 594.399,Z 234.066,A -85,B 0,C 180,E1 -1239.224,E2 -1239.224} C_VEL
LIN {X 0,Y 594.373,Z 234.07,A -85,B 0,C 180,E1 -1242.095,E2 -1242.095} C_VEL
LIN {X 0,Y 594.365,Z 234.069,A -85,B 0,C 180,E1 -1244.218,E2 -1244.218} C_VEL
LIN {X 0,Y 594.368,Z 234.069,A -85,B 0,C 180,E1 -1247.016,E2 -1247.016} C_VEL
LIN {X 0,Y 594.385,Z 234.071,A -85,B 0,C 180,E1 -1249.783,E2 -1249.783} C_VEL
LIN {X 0,Y 594.394,Z 234.063,A -85,B 0,C 180,E1 -1252.526,E2 -1252.526} C_VEL
LIN {X 0,Y 594.399,Z 234.071,A -85,B 0,C 180,E1 -1255.252,E2 -1255.252} C_VEL
LIN {X 0,Y 594.381,Z 234.067,A -85,B 0,C 180,E1 -1257.966,E2 -1257.966} C_VEL
LIN {X 0,Y 594.42,Z 234.062,A -85,B 0,C 180,E1 -1260.677,E2 -1260.677} C_VEL
LIN {X 0,Y 594.38,Z 234.073,A -85,B 0,C 180,E1 -1263.388,E2 -1263.388} C_VEL
LIN {X 0,Y 594.354,Z 234.069,A -85,B 0,C 180,E1 -1266.108,E2 -1266.108} C_VEL
LIN {X 0,Y 594.393,Z 234.07,A -85,B 0,C 180,E1 -1268.841,E2 -1268.841} C_VEL
LIN {X 0,Y 594.383,Z 234.067,A -85,B 0,C 180,E1 -1271.595,E2 -1271.595} C_VEL
LIN {X 0,Y 594.377,Z 234.067,A -85,B 0,C 180,E1 -1274.376,E2 -1274.376} C_VEL
LIN {X 0,Y 594.352,Z 234.073,A -85,B 0,C 180,E1 -1275.34,E2 -1275.34} C_VEL
LIN {X 0,Y 593.678,Z 234.156,A -85,B 0,C 180,E1 -1275.906,E2 -1275.906} C_VEL
LIN {X 0,Y 590.811,Z 234.519,A -85,B 0,C 180,E1 -1276.824,E2 -1276.824} C_VEL
LIN {X 0,Y 588.4,Z 234.814,A -85,B 0,C 180,E1 -1277.563,E2 -1277.563} C_VEL
LIN {X 0,Y 587.378,Z 234.939,A -85,B 0,C 180,E1 -1278.133,E2 -1278.133} C_VEL
LIN {X 0,Y 587.302,Z 234.949,A -85,B 0,C 180,E1 -1278.326,E2 -1278.326} C_VEL
LIN {X 0,Y 587.344,Z 234.949,A -85,B 0,C 180,E1 -1281.044,E2 -1281.044} C_VEL
LIN {X 0,Y 587.354,Z 234.943,A -85,B 0,C 180,E1 -1283.256,E2 -1283.256} C_VEL
LIN {X 0,Y 587.345,Z 234.945,A -85,B 0,C 180,E1 -1286.181,E2 -1286.181} C_VEL
LIN {X 0,Y 587.34,Z 234.945,A -85,B 0,C 180,E1 -1289.134,E2 -1289.134} C_VEL
LIN {X 0,Y 587.333,Z 234.944,A -85,B 0,C 180,E1 -1291.836,E2 -1291.836} C_VEL
LIN {X 0,Y 587.338,Z 234.95,A -85,B 0,C 180,E1 -1294.348,E2 -1294.348} C_VEL
LIN {X 0,Y 587.337,Z 234.949,A -85,B 0,C 180,E1 -1296.746,E2 -1296.746} C_VEL
LIN {X 0,Y 587.332,Z 234.943,A -85,B 0,C 180,E1 -1299.359,E2 -1299.359} C_VEL
LIN {X 0,Y 587.351,Z 234.947,A -85,B 0,C 180,E1 -1302.111,E2 -1302.111} C_VEL
LIN {X 0,Y 587.299,Z 234.949,A -85,B 0,C 180,E1 -1305.088,E2 -1305.088} C_VEL
LIN {X 0,Y 587.336,Z 234.949,A -85,B 0,C 180,E1 -1307.927,E2 -1307.927} C_VEL
LIN {X 0,Y 587.332,Z 234.948,A -85,B 0,C 180,E1 -1310.641,E2 -1310.641} C_VEL
LIN {X 0,Y 587.337,Z 234.945,A -85,B 0,C 180,E1 -1313.291,E2 -1313.291} C_VEL
LIN {X 0,Y 587.332,Z 235.041,A -85,B 0,C 180,E1 -1314.924,E2 -1314.924} C_VEL
LIN {X 0,Y 587.692,Z 239.391,A -85,B 0,C 180,E1 -1315.601,E2 -1315.601} C_VEL
LIN {X 0,Y 587.495,Z 256.942,A -85,B 0,C 180,E1 -1318.241,E2 -1318.241} C_VEL
LIN {X 0,Y 587.507,Z 266.986,A -85,B 0,C 180,E1 -1319.708,E2 -1319.708} C_VEL
LIN {X 0,Y 588.163,Z 271.451,A -85,B 0,C 180,E1 -1319.782,E2 -1319.782} C_VEL
LIN {X 0,Y 587.98,Z 403.739,A -85,B 0,C 180,E1 -1321.439,E2 -1321.439} C_VEL
LIN {X 0,Y 587.897,Z 418.097,A -85,B 0,C 180,E1 -1321.763,E2 -1321.763} C_VEL
LIN {X 0,Y 587.834,Z 431.802,A -85,B 0,C 180,E1 -1322.214,E2 -1322.214} C_VEL
LIN {X 0,Y 587.724,Z 444.786,A -85,B 0,C 180,E1 -1322.782,E2 -1322.782} C_VEL
LIN {X 0,Y 587.625,Z 456.872,A -85,B 0,C 180,E1 -1323.449,E2 -1323.449} C_VEL
LIN {X 0,Y 587.506,Z 469.352,A -85,B 0,C 180,E1 -1324.302,E2 -1324.302} C_VEL
LIN {X 0,Y 587.421,Z 480.621,A -85,B 0,C 180,E1 -1325.245,E2 -1325.245} C_VEL
LIN {X 0,Y 587.371,Z 489.916,A -85,B 0,C 180,E1 -1326.183,E2 -1326.183} C_VEL
LIN {X 0,Y 587.275,Z 499.203,A -85,B 0,C 180,E1 -1327.307,E2 -1327.307} C_VEL
LIN {X 0,Y 587.249,Z 506.682,A -85,B 0,C 180,E1 -1328.408,E2 -1328.408} C_VEL
LIN {X 0,Y 587.201,Z 513.73,A -85,B 0,C 180,E1 -1329.691,E2 -1329.691} C_VEL
LIN {X 0,Y 587.167,Z 519.36,A -85,B 0,C 180,E1 -1331.005,E2 -1331.005} C_VEL
LIN {X 0,Y 587.156,Z 522.264,A -85,B 0,C 180,E1 -1331.868,E2 -1331.868} C_VEL
LIN {X 0,Y 587.148,Z 525.843,A -85,B 0,C 180,E1 -1333.306,E2 -1333.306} C_VEL
LIN {X 0,Y 587.136,Z 527.895,A -85,B 0,C 180,E1 -1334.732,E2 -1334.732} C_VEL
LIN {X 0,Y 587.149,Z 528.482,A -85,B 0,C 180,E1 -1336.15,E2 -1336.15} C_VEL
LIN {X 0,Y 587.16,Z 527.671,A -85,B 0,C 180,E1 -1337.558,E2 -1337.558} C_VEL
LIN {X 0,Y 587.146,Z 525.477,A -85,B 0,C 180,E1 -1338.959,E2 -1338.959} C_VEL
LIN {X 0,Y 587.16,Z 521.857,A -85,B 0,C 180,E1 -1340.354,E2 -1340.354} C_VEL
LIN {X 0,Y 587.183,Z 516.731,A -85,B 0,C 180,E1 -1341.742,E2 -1341.742} C_VEL
LIN {X 0,Y 587.206,Z 511.778,A -85,B 0,C 180,E1 -1342.781,E2 -1342.781} C_VEL
LIN {X 0,Y 587.267,Z 504.699,A -85,B 0,C 180,E1 -1343.99,E2 -1343.99} C_VEL
LIN {X 0,Y 587.304,Z 495.988,A -85,B 0,C 180,E1 -1345.195,E2 -1345.195} C_VEL
LIN {X 0,Y 587.362,Z 486.926,A -85,B 0,C 180,E1 -1346.227,E2 -1346.227} C_VEL
LIN {X 0,Y 587.472,Z 475.975,A -85,B 0,C 180,E1 -1347.257,E2 -1347.257} C_VEL
LIN {X 0,Y 587.542,Z 464.898,A -85,B 0,C 180,E1 -1348.115,E2 -1348.115} C_VEL
LIN {X 0,Y 587.661,Z 452.724,A -85,B 0,C 180,E1 -1348.887,E2 -1348.887} C_VEL
LIN {X 0,Y 587.788,Z 439.15,A -85,B 0,C 180,E1 -1349.572,E2 -1349.572} C_VEL
LIN {X 0,Y 587.857,Z 425.958,A -85,B 0,C 180,E1 -1350.086,E2 -1350.086} C_VEL
LIN {X 0,Y 587.928,Z 411.571,A -85,B 0,C 180,E1 -1350.492,E2 -1350.492} C_VEL
LIN {X 0,Y 587.969,Z 397.313,A -85,B 0,C 180,E1 -1350.749,E2 -1350.749} C_VEL
LIN {X 0,Y 588.13,Z 270.389,A -85,B 0,C 180,E1 -1352.322,E2 -1352.322} C_VEL
LIN {X 0,Y 587.478,Z 266.663,A -85,B 0,C 180,E1 -1352.4,E2 -1352.4} C_VEL
LIN {X 0,Y 587.664,Z 248.271,A -85,B 0,C 180,E1 -1355.146,E2 -1355.146} C_VEL
LIN {X 0,Y 587.62,Z 236.408,A -85,B 0,C 180,E1 -1356.947,E2 -1356.947} C_VEL
LIN {X 0,Y 587.381,Z 234.944,A -85,B 0,C 180,E1 -1357.217,E2 -1357.217} C_VEL
LIN {X 0,Y 587.34,Z 234.947,A -85,B 0,C 180,E1 -1360.34,E2 -1360.34} C_VEL
LIN {X 0,Y 587.312,Z 234.947,A -85,B 0,C 180,E1 -1363.142,E2 -1363.142} C_VEL
LIN {X 0,Y 587.323,Z 234.948,A -85,B 0,C 180,E1 -1365.263,E2 -1365.263} C_VEL
LIN {X 0,Y 587.349,Z 234.945,A -85,B 0,C 180,E1 -1367.406,E2 -1367.406} C_VEL
LIN {X 0,Y 587.324,Z 234.947,A -85,B 0,C 180,E1 -1370.305,E2 -1370.305} C_VEL
LIN {X 0,Y 587.314,Z 234.949,A -85,B 0,C 180,E1 -1373.259,E2 -1373.259} C_VEL
LIN {X 0,Y 587.353,Z 234.943,A -85,B 0,C 180,E1 -1376.183,E2 -1376.183} C_VEL
LIN {X 0,Y 587.343,Z 234.945,A -85,B 0,C 180,E1 -1379.135,E2 -1379.135} C_VEL
LIN {X 0,Y 587.348,Z 234.947,A -85,B 0,C 180,E1 -1381.839,E2 -1381.839} C_VEL
LIN {X 0,Y 587.346,Z 234.942,A -85,B 0,C 180,E1 -1384.35,E2 -1384.35} C_VEL
LIN {X 0,Y 587.339,Z 234.943,A -85,B 0,C 180,E1 -1386.747,E2 -1386.747} C_VEL
LIN {X 0,Y 587.335,Z 234.953,A -85,B 0,C 180,E1 -1389.359,E2 -1389.359} C_VEL
LIN {X 0,Y 587.352,Z 234.942,A -85,B 0,C 180,E1 -1392.112,E2 -1392.112} C_VEL
LIN {X 0,Y 587.301,Z 234.954,A -85,B 0,C 180,E1 -1395.089,E2 -1395.089} C_VEL
LIN {X 0,Y 587.338,Z 234.944,A -85,B 0,C 180,E1 -1397.928,E2 -1397.928} C_VEL
LIN {X 0,Y 587.337,Z 234.945,A -85,B 0,C 180,E1 -1400.642,E2 -1400.642} C_VEL
LIN {X 0,Y 587.341,Z 234.95,A -85,B 0,C 180,E1 -1403.292,E2 -1403.292} C_VEL
LIN {X 0,Y 587.36,Z 234.941,A -85,B 0,C 180,E1 -1405.782,E2 -1405.782} C_VEL
LIN {X 0,Y 587.341,Z 234.943,A -85,B 0,C 180,E1 -1408.233,E2 -1408.233} C_VEL
LIN {X 0,Y 587.341,Z 234.95,A -85,B 0,C 180,E1 -1410.866,E2 -1410.866} C_VEL
LIN {X 0,Y 587.349,Z 234.942,A -85,B 0,C 180,E1 -1413.819,E2 -1413.819} C_VEL
LIN {X 0,Y 587.33,Z 234.944,A -85,B 0,C 180,E1 -1415.995,E2 -1415.995} C_VEL
LIN {X 0,Y 587.335,Z 234.952,A -85,B 0,C 180,E1 -1418.964,E2 -1418.964} C_VEL
LIN {X 0,Y 587.32,Z 234.945,A -85,B 0,C 180,E1 -1421.874,E2 -1421.874} C_VEL
LIN {X 0,Y 587.321,Z 234.945,A -85,B 0,C 180,E1 -1424.026,E2 -1424.026} C_VEL
LIN {X 0,Y 587.353,Z 234.943,A -85,B 0,C 180,E1 -1426.155,E2 -1426.155} C_VEL
LIN {X 0,Y 587.335,Z 234.949,A -85,B 0,C 180,E1 -1428.963,E2 -1428.963} C_VEL
LIN {X 0,Y 587.362,Z 234.94,A -85,B 0,C 180,E1 -1431.746,E2 -1431.746} C_VEL
LIN {X 0,Y 587.354,Z 234.95,A -85,B 0,C 180,E1 -1434.508,E2 -1434.508} C_VEL
LIN {X 0,Y 587.372,Z 234.939,A -85,B 0,C 180,E1 -1437.258,E2 -1437.258} C_VEL
LIN {X 0,Y 587.374,Z 234.941,A -85,B 0,C 180,E1 -1440.001,E2 -1440.001} C_VEL
LIN {X 0,Y 587.372,Z 234.944,A -85,B 0,C 180,E1 -1442.744,E2 -1442.744} C_VEL
LIN {X 0,Y 587.355,Z 234.941,A -85,B 0,C 180,E1 -1445.494,E2 -1445.494} C_VEL
LIN {X 0,Y 587.364,Z 234.949,A -85,B 0,C 180,E1 -1448.256,E2 -1448.256} C_VEL
LIN {X 0,Y 587.34,Z 234.943,A -85,B 0,C 180,E1 -1451.135,E2 -1451.135} C_VEL
LIN {X 0,Y 587.358,Z 234.95,A -85,B 0,C 180,E1 -1454.262,E2 -1454.262} C_VEL
LIN {X 0,Y 587.354,Z 234.941,A -85,B 0,C 180,E1 -1457.407,E2 -1457.407} C_VEL
LIN {X 0,Y 587.326,Z 234.951,A -85,B 0,C 180,E1 -1460.306,E2 -1460.306} C_VEL
LIN {X 0,Y 587.319,Z 234.945,A -85,B 0,C 180,E1 -1463.26,E2 -1463.26} C_VEL
LIN {X 0,Y 587.33,Z 234.946,A -85,B 0,C 180,E1 -1465.517,E2 -1465.517} C_VEL
LIN {X 0,Y 587.343,Z 234.95,A -85,B 0,C 180,E1 -1467.819,E2 -1467.819} C_VEL
LIN {X 0,Y 587.347,Z 234.943,A -85,B 0,C 180,E1 -1470.513,E2 -1470.513} C_VEL
LIN {X 0,Y 587.331,Z 234.947,A -85,B 0,C 180,E1 -1473.398,E2 -1473.398} C_VEL
LIN {X 0,Y 587.353,Z 234.95,A -85,B 0,C 180,E1 -1475.896,E2 -1475.896} C_VEL
LIN {X 0,Y 587.33,Z 234.945,A -85,B 0,C 180,E1 -1478.48,E2 -1478.48} C_VEL
LIN {X 0,Y 587.333,Z 234.945,A -85,B 0,C 180,E1 -1481.158,E2 -1481.158} C_VEL
LIN {X 0,Y 587.324,Z 234.948,A -85,B 0,C 180,E1 -1484.114,E2 -1484.114} C_VEL
LIN {X 0,Y 587.322,Z 234.946,A -85,B 0,C 180,E1 -1486.995,E2 -1486.995} C_VEL
LIN {X 0,Y 587.311,Z 234.953,A -85,B 0,C 180,E1 -1489.746,E2 -1489.746} C_VEL
LIN {X 0,Y 587.342,Z 234.942,A -85,B 0,C 180,E1 -1492.393,E2 -1492.393} C_VEL
LIN {X 0,Y 587.361,Z 234.945,A -85,B 0,C 180,E1 -1495.781,E2 -1495.781} C_VEL
LIN {X 0,Y 587.346,Z 234.943,A -85,B 0,C 180,E1 -1498.232,E2 -1498.232} C_VEL
LIN {X 0,Y 587.35,Z 234.945,A -85,B 0,C 180,E1 -1500.867,E2 -1500.867} C_VEL
LIN {X 0,Y 587.36,Z 234.945,A -85,B 0,C 180,E1 -1503.819,E2 -1503.819} C_VEL
LIN {X 0,Y 587.368,Z 235.091,A -85,B 0,C 180,E1 -1505.809,E2 -1505.809} C_VEL
LIN {X 0,Y 588.026,Z 239.319,A -85,B 0,C 180,E1 -1506.398,E2 -1506.398} C_VEL
LIN {X 0,Y 587.854,Z 261.928,A -85,B 0,C 180,E1 -1509.349,E2 -1509.349} C_VEL
LIN {X 0,Y 587.629,Z 285.949,A -85,B 0,C 180,E1 -1512.423,E2 -1512.423} C_VEL
LIN {X 0,Y 587.56,Z 295.576,A -85,B 0,C 180,E1 -1513.641,E2 -1513.641} C_VEL
LIN {X 0,Y 588.204,Z 299.638,A -85,B 0,C 180,E1 -1513.716,E2 -1513.716} C_VEL
LIN {X 0,Y 587.992,Z 433.898,A -85,B 0,C 180,E1 -1515.397,E2 -1515.397} C_VEL
LIN {X 0,Y 587.943,Z 448.314,A -85,B 0,C 180,E1 -1515.725,E2 -1515.725} C_VEL
LIN {X 0,Y 587.805,Z 462.844,A -85,B 0,C 180,E1 -1516.209,E2 -1516.209} C_VEL
LIN {X 0,Y 587.725,Z 475.643,A -85,B 0,C 180,E1 -1516.78,E2 -1516.78} C_VEL
LIN {X 0,Y 587.604,Z 488.101,A -85,B 0,C 180,E1 -1517.48,E2 -1517.48} C_VEL
LIN {X 0,Y 587.513,Z 500.641,A -85,B 0,C 180,E1 -1518.354,E2 -1518.354} C_VEL
LIN {X 0,Y 587.445,Z 511.837,A -85,B 0,C 180,E1 -1519.314,E2 -1519.314} C_VEL
LIN {X 0,Y 587.319,Z 521.852,A -85,B 0,C 180,E1 -1520.356,E2 -1520.356} C_VEL
LIN {X 0,Y 587.277,Z 530.172,A -85,B 0,C 180,E1 -1521.397,E2 -1521.397} C_VEL
LIN {X 0,Y 587.244,Z 538.126,A -85,B 0,C 180,E1 -1522.608,E2 -1522.608} C_VEL
LIN {X 0,Y 587.204,Z 544.527,A -85,B 0,C 180,E1 -1523.816,E2 -1523.816} C_VEL
LIN {X 0,Y 587.16,Z 548.961,A -85,B 0,C 180,E1 -1524.85,E2 -1524.85} C_VEL
LIN {X 0,Y 587.179,Z 552.442,A -85,B 0,C 180,E1 -1525.882,E2 -1525.882} C_VEL
LIN {X 0,Y 587.13,Z 555.831,A -85,B 0,C 180,E1 -1527.256,E2 -1527.256} C_VEL
LIN {X 0,Y 587.142,Z 557.832,A -85,B 0,C 180,E1 -1528.628,E2 -1528.628} C_VEL
LIN {X 0,Y 587.135,Z 558.5,A -85,B 0,C 180,E1 -1530,E2 -1530} C_VEL
LIN {X 0,Y 587.142,Z 557.832,A -85,B 0,C 180,E1 -1531.372,E2 -1531.372} C_VEL
LIN {X 0,Y 587.13,Z 555.833,A -85,B 0,C 180,E1 -1532.744,E2 -1532.744} C_VEL
LIN {X 0,Y 587.179,Z 552.444,A -85,B 0,C 180,E1 -1534.118,E2 -1534.118} C_VEL
LIN {X 0,Y 587.2,Z 547.569,A -85,B 0,C 180,E1 -1535.494,E2 -1535.494} C_VEL
LIN {X 0,Y 587.209,Z 541.053,A -85,B 0,C 180,E1 -1536.874,E2 -1536.874} C_VEL
LIN {X 0,Y 587.268,Z 533.801,A -85,B 0,C 180,E1 -1538.083,E2 -1538.083} C_VEL
LIN {X 0,Y 587.321,Z 524.825,A -85,B 0,C 180,E1 -1539.296,E2 -1539.296} C_VEL
LIN {X 0,Y 587.372,Z 515.394,A -85,B 0,C 180,E1 -1540.339,E2 -1540.339} C_VEL
LIN {X 0,Y 587.475,Z 505.032,A -85,B 0,C 180,E1 -1541.29,E2 -1541.29} C_VEL
LIN {X 0,Y 587.577,Z 493.436,A -85,B 0,C 180,E1 -1542.17,E2 -1542.17} C_VEL
LIN {X 0,Y 587.669,Z 480.654,A -85,B 0,C 180,E1 -1542.957,E2 -1542.957} C_VEL
LIN {X 0,Y 587.775,Z 468.167,A -85,B 0,C 180,E1 -1543.571,E2 -1543.571} C_VEL
LIN {X 0,Y 587.912,Z 454.618,A -85,B 0,C 180,E1 -1544.085,E2 -1544.085} C_VEL
LIN {X 0,Y 587.946,Z 440.983,A -85,B 0,C 180,E1 -1544.461,E2 -1544.461} C_VEL
LIN {X 0,Y 588.01,Z 426.632,A -85,B 0,C 180,E1 -1544.713,E2 -1544.713} C_VEL
LIN {X 0,Y 588.05,Z 298.31,A -85,B 0,C 180,E1 -1546.305,E2 -1546.305} C_VEL
LIN {X 0,Y 587.574,Z 295.489,A -85,B 0,C 180,E1 -1546.369,E2 -1546.369} C_VEL
LIN {X 0,Y 587.708,Z 274.644,A -85,B 0,C 180,E1 -1549.018,E2 -1549.018} C_VEL
LIN {X 0,Y 587.875,Z 254.811,A -85,B 0,C 180,E1 -1551.575,E2 -1551.575} C_VEL
LIN {X 0,Y 587.938,Z 237.908,A -85,B 0,C 180,E1 -1553.792,E2 -1553.792} C_VEL
LIN {X 0,Y 587.361,Z 234.948,A -85,B 0,C 180,E1 -1554.212,E2 -1554.212} C_VEL
LIN {X 0,Y 587.328,Z 234.949,A -85,B 0,C 180,E1 -1557.046,E2 -1557.046} C_VEL
LIN {X 0,Y 587.346,Z 234.943,A -85,B 0,C 180,E1 -1559.379,E2 -1559.379} C_VEL
LIN {X 0,Y 587.349,Z 234.943,A -85,B 0,C 180,E1 -1561.836,E2 -1561.836} C_VEL
LIN {X 0,Y 587.348,Z 234.951,A -85,B 0,C 180,E1 -1564.347,E2 -1564.347} C_VEL
LIN {X 0,Y 587.342,Z 234.943,A -85,B 0,C 180,E1 -1567.607,E2 -1567.607} C_VEL
LIN {X 0,Y 587.311,Z 234.956,A -85,B 0,C 180,E1 -1570.253,E2 -1570.253} C_VEL
LIN {X 0,Y 587.321,Z 234.946,A -85,B 0,C 180,E1 -1573.005,E2 -1573.005} C_VEL
LIN {X 0,Y 587.323,Z 234.949,A -85,B 0,C 180,E1 -1575.886,E2 -1575.886} C_VEL
LIN {X 0,Y 587.333,Z 234.945,A -85,B 0,C 180,E1 -1578.842,E2 -1578.842} C_VEL
LIN {X 0,Y 587.33,Z 234.946,A -85,B 0,C 180,E1 -1581.52,E2 -1581.52} C_VEL
LIN {X 0,Y 587.347,Z 234.944,A -85,B 0,C 180,E1 -1584.454,E2 -1584.454} C_VEL
LIN {X 0,Y 587.334,Z 234.944,A -85,B 0,C 180,E1 -1586.887,E2 -1586.887} C_VEL
LIN {X 0,Y 587.346,Z 234.944,A -85,B 0,C 180,E1 -1589.486,E2 -1589.486} C_VEL
LIN {X 0,Y 587.345,Z 234.945,A -85,B 0,C 180,E1 -1592.306,E2 -1592.306} C_VEL
LIN {X 0,Y 587.345,Z 234.944,A -85,B 0,C 180,E1 -1595.241,E2 -1595.241} C_VEL
LIN {X 0,Y 587.316,Z 234.949,A -85,B 0,C 180,E1 -1598.225,E2 -1598.225} C_VEL
LIN {X 0,Y 587.343,Z 234.944,A -85,B 0,C 180,E1 -1601.15,E2 -1601.15} C_VEL
LIN {X 0,Y 587.35,Z 234.946,A -85,B 0,C 180,E1 -1603.31,E2 -1603.31} C_VEL
LIN {X 0,Y 587.354,Z 234.943,A -85,B 0,C 180,E1 -1606.153,E2 -1606.153} C_VEL
LIN {X 0,Y 587.338,Z 234.944,A -85,B 0,C 180,E1 -1608.962,E2 -1608.962} C_VEL
LIN {X 0,Y 587.362,Z 234.945,A -85,B 0,C 180,E1 -1611.744,E2 -1611.744} C_VEL
LIN {X 0,Y 587.354,Z 234.941,A -85,B 0,C 180,E1 -1614.506,E2 -1614.506} C_VEL
LIN {X 0,Y 587.373,Z 234.947,A -85,B 0,C 180,E1 -1617.256,E2 -1617.256} C_VEL
LIN {X 0,Y 587.367,Z 234.94,A -85,B 0,C 180,E1 -1619.999,E2 -1619.999} C_VEL
LIN {X 0,Y 587.374,Z 234.941,A -85,B 0,C 180,E1 -1622.742,E2 -1622.742} C_VEL
LIN {X 0,Y 587.351,Z 234.946,A -85,B 0,C 180,E1 -1625.492,E2 -1625.492} C_VEL
LIN {X 0,Y 587.358,Z 234.941,A -85,B 0,C 180,E1 -1628.254,E2 -1628.254} C_VEL
LIN {X 0,Y 587.35,Z 234.95,A -85,B 0,C 180,E1 -1631.141,E2 -1631.141} C_VEL
LIN {X 0,Y 587.351,Z 234.942,A -85,B 0,C 180,E1 -1634.26,E2 -1634.26} C_VEL
LIN {X 0,Y 587.339,Z 234.945,A -85,B 0,C 180,E1 -1637.405,E2 -1637.405} C_VEL
LIN {X 0,Y 587.302,Z 234.949,A -85,B 0,C 180,E1 -1638.326,E2 -1638.326} C_VEL
LIN {X 0,Y 586.659,Z 235.038,A -85,B 0,C 180,E1 -1638.898,E2 -1638.898} C_VEL
LIN {X 0,Y 583.83,Z 235.39,A -85,B 0,C 180,E1 -1639.826,E2 -1639.826} C_VEL
LIN {X 0,Y 581.418,Z 235.689,A -85,B 0,C 180,E1 -1640.574,E2 -1640.574} C_VEL
LIN {X 0,Y 580.368,Z 235.817,A -85,B 0,C 180,E1 -1641.15,E2 -1641.15} C_VEL
LIN {X 0,Y 580.276,Z 235.825,A -85,B 0,C 180,E1 -1641.345,E2 -1641.345} C_VEL
LIN {X 0,Y 580.29,Z 235.821,A -85,B 0,C 180,E1 -1643.556,E2 -1643.556} C_VEL
LIN {X 0,Y 580.277,Z 235.827,A -85,B 0,C 180,E1 -1646.334,E2 -1646.334} C_VEL
LIN {X 0,Y 580.284,Z 235.826,A -85,B 0,C 180,E1 -1648.975,E2 -1648.975} C_VEL
LIN {X 0,Y 580.265,Z 235.824,A -85,B 0,C 180,E1 -1651.385,E2 -1651.385} C_VEL
LIN {X 0,Y 580.304,Z 235.82,A -85,B 0,C 180,E1 -1653.854,E2 -1653.854} C_VEL
LIN {X 0,Y 580.278,Z 235.83,A -85,B 0,C 180,E1 -1656.401,E2 -1656.401} C_VEL
LIN {X 0,Y 580.294,Z 235.821,A -85,B 0,C 180,E1 -1659.187,E2 -1659.187} C_VEL
LIN {X 0,Y 580.298,Z 235.822,A -85,B 0,C 180,E1 -1661.765,E2 -1661.765} C_VEL
LIN {X 0,Y 580.252,Z 235.831,A -85,B 0,C 180,E1 -1664.625,E2 -1664.625} C_VEL
LIN {X 0,Y 580.265,Z 235.825,A -85,B 0,C 180,E1 -1667.294,E2 -1667.294} C_VEL
LIN {X 0,Y 580.284,Z 235.831,A -85,B 0,C 180,E1 -1670.068,E2 -1670.068} C_VEL
LIN {X 0,Y 580.285,Z 235.824,A -85,B 0,C 180,E1 -1673.065,E2 -1673.065} C_VEL
LIN {X 0,Y 580.283,Z 235.988,A -85,B 0,C 180,E1 -1674.802,E2 -1674.802} C_VEL
LIN {X 0,Y 580.758,Z 239.572,A -85,B 0,C 180,E1 -1675.373,E2 -1675.373} C_VEL
LIN {X 0,Y 580.566,Z 256.305,A -85,B 0,C 180,E1 -1677.925,E2 -1677.925} C_VEL
LIN {X 0,Y 580.504,Z 266.865,A -85,B 0,C 180,E1 -1679.503,E2 -1679.503} C_VEL
LIN {X 0,Y 581.372,Z 272.626,A -85,B 0,C 180,E1 -1679.602,E2 -1679.602} C_VEL
LIN {X 0,Y 581.116,Z 404.001,A -85,B 0,C 180,E1 -1681.267,E2 -1681.267} C_VEL
LIN {X 0,Y 581.003,Z 418.251,A -85,B 0,C 180,E1 -1681.594,E2 -1681.594} C_VEL
LIN {X 0,Y 580.941,Z 431.83,A -85,B 0,C 180,E1 -1682.048,E2 -1682.048} C_VEL
LIN {X 0,Y 580.785,Z 444.866,A -85,B 0,C 180,E1 -1682.624,E2 -1682.624} C_VEL
LIN {X 0,Y 580.654,Z 456.93,A -85,B 0,C 180,E1 -1683.299,E2 -1683.299} C_VEL
LIN {X 0,Y 580.513,Z 469.403,A -85,B 0,C 180,E1 -1684.162,E2 -1684.162} C_VEL
LIN {X 0,Y 580.416,Z 480.781,A -85,B 0,C 180,E1 -1685.128,E2 -1685.128} C_VEL
LIN {X 0,Y 580.321,Z 489.946,A -85,B 0,C 180,E1 -1686.065,E2 -1686.065} C_VEL
LIN {X 0,Y 580.218,Z 499.168,A -85,B 0,C 180,E1 -1687.195,E2 -1687.195} C_VEL
LIN {X 0,Y 580.198,Z 506.708,A -85,B 0,C 180,E1 -1688.319,E2 -1688.319} C_VEL
LIN {X 0,Y 580.121,Z 512.842,A -85,B 0,C 180,E1 -1689.432,E2 -1689.432} C_VEL
LIN {X 0,Y 580.116,Z 517.801,A -85,B 0,C 180,E1 -1690.54,E2 -1690.54} C_VEL
LIN {X 0,Y 580.064,Z 521.722,A -85,B 0,C 180,E1 -1691.639,E2 -1691.639} C_VEL
LIN {X 0,Y 580.05,Z 525.479,A -85,B 0,C 180,E1 -1693.095,E2 -1693.095} C_VEL
LIN {X 0,Y 580.032,Z 527.703,A -85,B 0,C 180,E1 -1694.54,E2 -1694.54} C_VEL
LIN {X 0,Y 580.061,Z 528.491,A -85,B 0,C 180,E1 -1695.977,E2 -1695.977} C_VEL
LIN {X 0,Y 580.048,Z 527.866,A -85,B 0,C 180,E1 -1697.403,E2 -1697.403} C_VEL
LIN {X 0,Y 580.057,Z 525.833,A -85,B 0,C 180,E1 -1698.822,E2 -1698.822} C_VEL
LIN {X 0,Y 580.062,Z 522.38,A -85,B 0,C 180,E1 -1700.234,E2 -1700.234} C_VEL
LIN {X 0,Y 580.105,Z 517.429,A -85,B 0,C 180,E1 -1701.641,E2 -1701.641} C_VEL
LIN {X 0,Y 580.119,Z 512.666,A -85,B 0,C 180,E1 -1702.692,E2 -1702.692} C_VEL
LIN {X 0,Y 580.197,Z 505.79,A -85,B 0,C 180,E1 -1703.916,E2 -1703.916} C_VEL
LIN {X 0,Y 580.245,Z 497.311,A -85,B 0,C 180,E1 -1705.137,E2 -1705.137} C_VEL
LIN {X 0,Y 580.319,Z 488.502,A -85,B 0,C 180,E1 -1706.181,E2 -1706.181} C_VEL
LIN {X 0,Y 580.452,Z 477.892,A -85,B 0,C 180,E1 -1707.224,E2 -1707.224} C_VEL
LIN {X 0,Y 580.544,Z 466.077,A -85,B 0,C 180,E1 -1708.179,E2 -1708.179} C_VEL
LIN {X 0,Y 580.705,Z 454.185,A -85,B 0,C 180,E1 -1708.96,E2 -1708.96} C_VEL
LIN {X 0,Y 580.872,Z 440.977,A -85,B 0,C 180,E1 -1709.653,E2 -1709.653} C_VEL
LIN {X 0,Y 580.963,Z 427.093,A -85,B 0,C 180,E1 -1710.217,E2 -1710.217} C_VEL
LIN {X 0,Y 581.049,Z 412.282,A -85,B 0,C 180,E1 -1710.65,E2 -1710.65} C_VEL
LIN {X 0,Y 581.113,Z 398.458,A -85,B 0,C 180,E1 -1710.91,E2 -1710.91} C_VEL
LIN {X 0,Y 581.266,Z 271.001,A -85,B 0,C 180,E1 -1712.512,E2 -1712.512} C_VEL
LIN {X 0,Y 580.489,Z 266.663,A -85,B 0,C 180,E1 -1712.602,E2 -1712.602} C_VEL
LIN {X 0,Y 580.673,Z 248.289,A -85,B 0,C 180,E1 -1715.382,E2 -1715.382} C_VEL
LIN {X 0,Y 580.644,Z 237.568,A -85,B 0,C 180,E1 -1717.03,E2 -1717.03} C_VEL
LIN {X 0,Y 580.33,Z 235.823,A -85,B 0,C 180,E1 -1717.349,E2 -1717.349} C_VEL
LIN {X 0,Y 580.298,Z 235.823,A -85,B 0,C 180,E1 -1720.467,E2 -1720.467} C_VEL
LIN {X 0,Y 580.27,Z 235.826,A -85,B 0,C 180,E1 -1723.304,E2 -1723.304} C_VEL
LIN {X 0,Y 580.288,Z 235.826,A -85,B 0,C 180,E1 -1725.453,E2 -1725.453} C_VEL
LIN {X 0,Y 580.295,Z 235.827,A -85,B 0,C 180,E1 -1727.624,E2 -1727.624} C_VEL
LIN {X 0,Y 580.296,Z 235.83,A -85,B 0,C 180,E1 -1729.822,E2 -1729.822} C_VEL
LIN {X 0,Y 580.264,Z 235.829,A -85,B 0,C 180,E1 -1732.053,E2 -1732.053} C_VEL
LIN {X 0,Y 580.298,Z 235.821,A -85,B 0,C 180,E1 -1735.08,E2 -1735.08} C_VEL
LIN {X 0,Y 580.307,Z 235.825,A -85,B 0,C 180,E1 -1737.864,E2 -1737.864} C_VEL
LIN {X 0,Y 580.286,Z 235.821,A -85,B 0,C 180,E1 -1740.698,E2 -1740.698} C_VEL
LIN {X 0,Y 580.296,Z 235.827,A -85,B 0,C 180,E1 -1743.318,E2 -1743.318} C_VEL
LIN {X 0,Y 580.313,Z 235.823,A -85,B 0,C 180,E1 -1745.768,E2 -1745.768} C_VEL
LIN {X 0,Y 580.276,Z 235.823,A -85,B 0,C 180,E1 -1748.146,E2 -1748.146} C_VEL
LIN {X 0,Y 580.307,Z 235.821,A -85,B 0,C 180,E1 -1750.842,E2 -1750.842} C_VEL
LIN {X 0,Y 580.277,Z 235.827,A -85,B 0,C 180,E1 -1753.657,E2 -1753.657} C_VEL
LIN {X 0,Y 580.277,Z 235.823,A -85,B 0,C 180,E1 -1756.608,E2 -1756.608} C_VEL
LIN {X 0,Y 580.306,Z 235.828,A -85,B 0,C 180,E1 -1759.159,E2 -1759.159} C_VEL
LIN {X 0,Y 580.279,Z 235.823,A -85,B 0,C 180,E1 -1761.927,E2 -1761.927} C_VEL
LIN {X 0,Y 580.297,Z 235.821,A -85,B 0,C 180,E1 -1764.458,E2 -1764.458} C_VEL
LIN {X 0,Y 580.279,Z 235.83,A -85,B 0,C 180,E1 -1766.976,E2 -1766.976} C_VEL
LIN {X 0,Y 580.299,Z 235.824,A -85,B 0,C 180,E1 -1769.427,E2 -1769.427} C_VEL
LIN {X 0,Y 580.307,Z 235.819,A -85,B 0,C 180,E1 -1772.137,E2 -1772.137} C_VEL
LIN {X 0,Y 580.297,Z 235.83,A -85,B 0,C 180,E1 -1774.921,E2 -1774.921} C_VEL
LIN {X 0,Y 580.264,Z 235.824,A -85,B 0,C 180,E1 -1777.948,E2 -1777.948} C_VEL
LIN {X 0,Y 580.306,Z 235.828,A -85,B 0,C 180,E1 -1780.915,E2 -1780.915} C_VEL
LIN {X 0,Y 580.274,Z 235.823,A -85,B 0,C 180,E1 -1783.827,E2 -1783.827} C_VEL
LIN {X 0,Y 580.274,Z 235.833,A -85,B 0,C 180,E1 -1786.697,E2 -1786.697} C_VEL
LIN {X 0,Y 580.295,Z 235.82,A -85,B 0,C 180,E1 -1789.534,E2 -1789.534} C_VEL
LIN {X 0,Y 580.324,Z 235.822,A -85,B 0,C 180,E1 -1792.346,E2 -1792.346} C_VEL
LIN {X 0,Y 580.332,Z 235.818,A -85,B 0,C 180,E1 -1795.138,E2 -1795.138} C_VEL
LIN {X 0,Y 580.33,Z 235.817,A -85,B 0,C 180,E1 -1797.919,E2 -1797.919} C_VEL
LIN {X 0,Y 580.358,Z 235.819,A -85,B 0,C 180,E1 -1800.695,E2 -1800.695} C_VEL
LIN {X 0,Y 580.281,Z 235.822,A -85,B 0,C 180,E1 -1803.473,E2 -1803.473} C_VEL
LIN {X 0,Y 580.32,Z 235.817,A -85,B 0,C 180,E1 -1805.561,E2 -1805.561} C_VEL
LIN {X 0,Y 580.327,Z 235.826,A -85,B 0,C 180,E1 -1808.357,E2 -1808.357} C_VEL
LIN {X 0,Y 580.292,Z 235.821,A -85,B 0,C 180,E1 -1811.192,E2 -1811.192} C_VEL
LIN {X 0,Y 580.321,Z 235.823,A -85,B 0,C 180,E1 -1814.018,E2 -1814.018} C_VEL
LIN {X 0,Y 580.306,Z 235.819,A -85,B 0,C 180,E1 -1816.915,E2 -1816.915} C_VEL
LIN {X 0,Y 580.301,Z 235.824,A -85,B 0,C 180,E1 -1819.823,E2 -1819.823} C_VEL
LIN {X 0,Y 580.29,Z 235.822,A -85,B 0,C 180,E1 -1822.803,E2 -1822.803} C_VEL
LIN {X 0,Y 580.302,Z 235.819,A -85,B 0,C 180,E1 -1825.081,E2 -1825.081} C_VEL
LIN {X 0,Y 580.296,Z 235.827,A -85,B 0,C 180,E1 -1828.186,E2 -1828.186} C_VEL
LIN {X 0,Y 580.295,Z 235.821,A -85,B 0,C 180,E1 -1830.698,E2 -1830.698} C_VEL
LIN {X 0,Y 580.299,Z 235.822,A -85,B 0,C 180,E1 -1833.317,E2 -1833.317} C_VEL
LIN {X 0,Y 580.322,Z 235.826,A -85,B 0,C 180,E1 -1835.768,E2 -1835.768} C_VEL
LIN {X 0,Y 580.286,Z 235.826,A -85,B 0,C 180,E1 -1838.147,E2 -1838.147} C_VEL
LIN {X 0,Y 580.296,Z 235.82,A -85,B 0,C 180,E1 -1840.844,E2 -1840.844} C_VEL
LIN {X 0,Y 580.276,Z 235.832,A -85,B 0,C 180,E1 -1843.659,E2 -1843.659} C_VEL
LIN {X 0,Y 580.284,Z 235.821,A -85,B 0,C 180,E1 -1846.609,E2 -1846.609} C_VEL
LIN {X 0,Y 580.297,Z 235.823,A -85,B 0,C 180,E1 -1849.157,E2 -1849.157} C_VEL
LIN {X 0,Y 580.288,Z 235.825,A -85,B 0,C 180,E1 -1851.928,E2 -1851.928} C_VEL
LIN {X 0,Y 580.251,Z 235.826,A -85,B 0,C 180,E1 -1854.453,E2 -1854.453} C_VEL
LIN {X 0,Y 580.292,Z 235.823,A -85,B 0,C 180,E1 -1856.976,E2 -1856.976} C_VEL
LIN {X 0,Y 580.295,Z 235.831,A -85,B 0,C 180,E1 -1859.426,E2 -1859.426} C_VEL
LIN {X 0,Y 580.298,Z 235.822,A -85,B 0,C 180,E1 -1862.142,E2 -1862.142} C_VEL
LIN {X 0,Y 580.323,Z 235.827,A -85,B 0,C 180,E1 -1865.27,E2 -1865.27} C_VEL
LIN {X 0,Y 580.321,Z 235.932,A -85,B 0,C 180,E1 -1865.622,E2 -1865.622} C_VEL
LIN {X 0,Y 581.146,Z 240.72,A -85,B 0,C 180,E1 -1866.291,E2 -1866.291} C_VEL
LIN {X 0,Y 580.927,Z 261.928,A -85,B 0,C 180,E1 -1869.091,E2 -1869.091} C_VEL
LIN {X 0,Y 580.714,Z 284.536,A -85,B 0,C 180,E1 -1872.025,E2 -1872.025} C_VEL
LIN {X 0,Y 580.584,Z 295.62,A -85,B 0,C 180,E1 -1873.445,E2 -1873.445} C_VEL
LIN {X 0,Y 581.391,Z 301.427,A -85,B 0,C 180,E1 -1873.542,E2 -1873.542} C_VEL
LIN {X 0,Y 581.123,Z 433.897,A -85,B 0,C 180,E1 -1875.221,E2 -1875.221} C_VEL
LIN {X 0,Y 581.022,Z 448.021,A -85,B 0,C 180,E1 -1875.543,E2 -1875.543} C_VEL
LIN {X 0,Y 580.906,Z 461.717,A -85,B 0,C 180,E1 -1875.998,E2 -1875.998} C_VEL
LIN {X 0,Y 580.786,Z 475.646,A -85,B 0,C 180,E1 -1876.619,E2 -1876.619} C_VEL
LIN {X 0,Y 580.656,Z 488.103,A -85,B 0,C 180,E1 -1877.328,E2 -1877.328} C_VEL
LIN {X 0,Y 580.525,Z 500.644,A -85,B 0,C 180,E1 -1878.212,E2 -1878.212} C_VEL
LIN {X 0,Y 580.441,Z 511.894,A -85,B 0,C 180,E1 -1879.189,E2 -1879.189} C_VEL
LIN {X 0,Y 580.276,Z 521.852,A -85,B 0,C 180,E1 -1880.238,E2 -1880.238} C_VEL
LIN {X 0,Y 580.241,Z 530.173,A -85,B 0,C 180,E1 -1881.292,E2 -1881.292} C_VEL
LIN {X 0,Y 580.166,Z 538.127,A -85,B 0,C 180,E1 -1882.518,E2 -1882.518} C_VEL
LIN {X 0,Y 580.103,Z 544.528,A -85,B 0,C 180,E1 -1883.74,E2 -1883.74} C_VEL
LIN {X 0,Y 580.078,Z 548.961,A -85,B 0,C 180,E1 -1884.787,E2 -1884.787} C_VEL
LIN {X 0,Y 580.102,Z 552.443,A -85,B 0,C 180,E1 -1885.831,E2 -1885.831} C_VEL
LIN {X 0,Y 580.041,Z 555.832,A -85,B 0,C 180,E1 -1887.222,E2 -1887.222} C_VEL
LIN {X 0,Y 580.041,Z 557.832,A -85,B 0,C 180,E1 -1888.611,E2 -1888.611} C_VEL
LIN {X 0,Y 580.036,Z 558.5,A -85,B 0,C 180,E1 -1890,E2 -1890} C_VEL
LIN {X 0,Y 580.041,Z 557.833,A -85,B 0,C 180,E1 -1891.388,E2 -1891.388} C_VEL
LIN {X 0,Y 580.041,Z 555.833,A -85,B 0,C 180,E1 -1892.778,E2 -1892.778} C_VEL
LIN {X 0,Y 580.102,Z 552.445,A -85,B 0,C 180,E1 -1894.168,E2 -1894.168} C_VEL
LIN {X 0,Y 580.128,Z 547.569,A -85,B 0,C 180,E1 -1895.561,E2 -1895.561} C_VEL
LIN {X 0,Y 580.141,Z 541.054,A -85,B 0,C 180,E1 -1896.958,E2 -1896.958} C_VEL
LIN {X 0,Y 580.192,Z 533.802,A -85,B 0,C 180,E1 -1898.182,E2 -1898.182} C_VEL
LIN {X 0,Y 580.284,Z 524.825,A -85,B 0,C 180,E1 -1899.41,E2 -1899.41} C_VEL
LIN {X 0,Y 580.356,Z 515.395,A -85,B 0,C 180,E1 -1900.465,E2 -1900.465} C_VEL
LIN {X 0,Y 580.476,Z 505.324,A -85,B 0,C 180,E1 -1901.404,E2 -1901.404} C_VEL
LIN {X 0,Y 580.617,Z 493.438,A -85,B 0,C 180,E1 -1902.318,E2 -1902.318} C_VEL
LIN {X 0,Y 580.728,Z 480.652,A -85,B 0,C 180,E1 -1903.115,E2 -1903.115} C_VEL
LIN {X 0,Y 580.851,Z 468.164,A -85,B 0,C 180,E1 -1903.736,E2 -1903.736} C_VEL
LIN {X 0,Y 581.016,Z 455.204,A -85,B 0,C 180,E1 -1904.235,E2 -1904.235} C_VEL
LIN {X 0,Y 581.083,Z 441.19,A -85,B 0,C 180,E1 -1904.63,E2 -1904.63} C_VEL
LIN {X 0,Y 581.158,Z 426.632,A -85,B 0,C 180,E1 -1904.89,E2 -1904.89} C_VEL
LIN {X 0,Y 581.315,Z 299.65,A -85,B 0,C 180,E1 -1906.483,E2 -1906.483} C_VEL
LIN {X 0,Y 580.595,Z 295.489,A -85,B 0,C 180,E1 -1906.572,E2 -1906.572} C_VEL
LIN {X 0,Y 580.787,Z 274.371,A -85,B 0,C 180,E1 -1909.289,E2 -1909.289} C_VEL
LIN {X 0,Y 581.017,Z 253.451,A -85,B 0,C 180,E1 -1912.022,E2 -1912.022} C_VEL
LIN {X 0,Y 581.042,Z 239.285,A -85,B 0,C 180,E1 -1913.903,E2 -1913.903} C_VEL
LIN {X 0,Y 580.329,Z 235.826,A -85,B 0,C 180,E1 -1914.409,E2 -1914.409} C_VEL
LIN {X 0,Y 580.287,Z 235.823,A -85,B 0,C 180,E1 -1917.401,E2 -1917.401} C_VEL
LIN {X 0,Y 580.287,Z 235.823,A -85,B 0,C 180,E1 -1919.772,E2 -1919.772} C_VEL
LIN {X 0,Y 580.3,Z 235.826,A -85,B 0,C 180,E1 -1922.2,E2 -1922.2} C_VEL
LIN {X 0,Y 580.289,Z 235.829,A -85,B 0,C 180,E1 -1924.695,E2 -1924.695} C_VEL
LIN {X 0,Y 580.296,Z 235.821,A -85,B 0,C 180,E1 -1927.268,E2 -1927.268} C_VEL
LIN {X 0,Y 580.29,Z 235.831,A -85,B 0,C 180,E1 -1930.27,E2 -1930.27} C_VEL
LIN {X 0,Y 580.28,Z 235.826,A -85,B 0,C 180,E1 -1932.705,E2 -1932.705} C_VEL
LIN {X 0,Y 580.266,Z 235.825,A -85,B 0,C 180,E1 -1935.608,E2 -1935.608} C_VEL
LIN {X 0,Y 580.31,Z 235.828,A -85,B 0,C 180,E1 -1938.233,E2 -1938.233} C_VEL
LIN {X 0,Y 580.286,Z 235.822,A -85,B 0,C 180,E1 -1940.965,E2 -1940.965} C_VEL
LIN {X 0,Y 580.292,Z 235.823,A -85,B 0,C 180,E1 -1943.598,E2 -1943.598} C_VEL
LIN {X 0,Y 580.314,Z 235.826,A -85,B 0,C 180,E1 -1946.145,E2 -1946.145} C_VEL
LIN {X 0,Y 580.284,Z 235.822,A -85,B 0,C 180,E1 -1948.614,E2 -1948.614} C_VEL
LIN {X 0,Y 580.288,Z 235.821,A -85,B 0,C 180,E1 -1951.023,E2 -1951.023} C_VEL
LIN {X 0,Y 580.285,Z 235.828,A -85,B 0,C 180,E1 -1953.665,E2 -1953.665} C_VEL
LIN {X 0,Y 580.295,Z 235.828,A -85,B 0,C 180,E1 -1955.683,E2 -1955.683} C_VEL
LIN {X 0,Y 580.267,Z 235.831,A -85,B 0,C 180,E1 -1957.946,E2 -1957.946} C_VEL
LIN {X 0,Y 580.311,Z 235.819,A -85,B 0,C 180,E1 -1960.913,E2 -1960.913} C_VEL
LIN {X 0,Y 580.277,Z 235.829,A -85,B 0,C 180,E1 -1963.825,E2 -1963.825} C_VEL
LIN {X 0,Y 580.274,Z 235.823,A -85,B 0,C 180,E1 -1966.695,E2 -1966.695} C_VEL
LIN {X 0,Y 580.295,Z 235.83,A -85,B 0,C 180,E1 -1969.532,E2 -1969.532} C_VEL
LIN {X 0,Y 580.324,Z 235.816,A -85,B 0,C 180,E1 -1972.344,E2 -1972.344} C_VEL
LIN {X 0,Y 580.337,Z 235.821,A -85,B 0,C 180,E1 -1975.136,E2 -1975.136} C_VEL
LIN {X 0,Y 580.324,Z 235.818,A -85,B 0,C 180,E1 -1977.917,E2 -1977.917} C_VEL
LIN {X 0,Y 580.359,Z 235.814,A -85,B 0,C 180,E1 -1980.693,E2 -1980.693} C_VEL
LIN {X 0,Y 580.281,Z 235.828,A -85,B 0,C 180,E1 -1983.471,E2 -1983.471} C_VEL
LIN {X 0,Y 580.316,Z 235.821,A -85,B 0,C 180,E1 -1985.559,E2 -1985.559} C_VEL
LIN {X 0,Y 580.323,Z 235.818,A -85,B 0,C 180,E1 -1988.355,E2 -1988.355} C_VEL
LIN {X 0,Y 580.321,Z 235.824,A -85,B 0,C 180,E1 -1991.207,E2 -1991.207} C_VEL
LIN {X 0,Y 580.302,Z 235.82,A -85,B 0,C 180,E1 -1994.338,E2 -1994.338} C_VEL
LIN {X 0,Y 580.302,Z 235.829,A -85,B 0,C 180,E1 -1996.914,E2 -1996.914} C_VEL
LIN {X 0,Y 580.296,Z 235.82,A -85,B 0,C 180,E1 -1999.821,E2 -1999.821} C_VEL
LIN {X 0,Y 580.276,Z 235.825,A -85,B 0,C 180,E1 -2001.345,E2 -2001.345} C_VEL
LIN {X 0,Y 579.585,Z 235.911,A -85,B 0,C 180,E1 -2001.925,E2 -2001.925} C_VEL
LIN {X 0,Y 576.713,Z 236.275,A -85,B 0,C 180,E1 -2002.865,E2 -2002.865} C_VEL
LIN {X 0,Y 574.316,Z 236.568,A -85,B 0,C 180,E1 -2003.621,E2 -2003.621} C_VEL
LIN {X 0,Y 573.311,Z 236.692,A -85,B 0,C 180,E1 -2004.206,E2 -2004.206} C_VEL
LIN {X 0,Y 573.241,Z 236.703,A -85,B 0,C 180,E1 -2004.403,E2 -2004.403} C_VEL
LIN {X 0,Y 573.237,Z 236.705,A -85,B 0,C 180,E1 -2006.975,E2 -2006.975} C_VEL
LIN {X 0,Y 573.24,Z 236.699,A -85,B 0,C 180,E1 -2009.489,E2 -2009.489} C_VEL
LIN {X 0,Y 573.241,Z 236.708,A -85,B 0,C 180,E1 -2012.644,E2 -2012.644} C_VEL
LIN {X 0,Y 573.24,Z 236.699,A -85,B 0,C 180,E1 -2015.184,E2 -2015.184} C_VEL
LIN {X 0,Y 573.222,Z 236.703,A -85,B 0,C 180,E1 -2017.807,E2 -2017.807} C_VEL
LIN {X 0,Y 573.253,Z 236.706,A -85,B 0,C 180,E1 -2020.528,E2 -2020.528} C_VEL
LIN {X 0,Y 573.236,Z 236.7,A -85,B 0,C 180,E1 -2023.357,E2 -2023.357} C_VEL
LIN {X 0,Y 573.236,Z 236.709,A -85,B 0,C 180,E1 -2026.33,E2 -2026.33} C_VEL
LIN {X 0,Y 573.258,Z 236.699,A -85,B 0,C 180,E1 -2029.477,E2 -2029.477} C_VEL
LIN {X 0,Y 573.222,Z 236.712,A -85,B 0,C 180,E1 -2032.193,E2 -2032.193} C_VEL
LIN {X 0,Y 573.25,Z 236.831,A -85,B 0,C 180,E1 -2034.655,E2 -2034.655} C_VEL
LIN {X 0,Y 573.794,Z 241.624,A -85,B 0,C 180,E1 -2035.431,E2 -2035.431} C_VEL
LIN {X 0,Y 573.561,Z 258.009,A -85,B 0,C 180,E1 -2037.958,E2 -2037.958} C_VEL
LIN {X 0,Y 573.525,Z 266.867,A -85,B 0,C 180,E1 -2039.296,E2 -2039.296} C_VEL
LIN {X 0,Y 574.547,Z 272.542,A -85,B 0,C 180,E1 -2039.399,E2 -2039.399} C_VEL
LIN {X 0,Y 574.276,Z 402.983,A -85,B 0,C 180,E1 -2041.068,E2 -2041.068} C_VEL
LIN {X 0,Y 574.159,Z 417.188,A -85,B 0,C 180,E1 -2041.387,E2 -2041.387} C_VEL
LIN {X 0,Y 574.035,Z 431.241,A -85,B 0,C 180,E1 -2041.853,E2 -2041.853} C_VEL
LIN {X 0,Y 573.908,Z 443.04,A -85,B 0,C 180,E1 -2042.367,E2 -2042.367} C_VEL
LIN {X 0,Y 573.727,Z 455.448,A -85,B 0,C 180,E1 -2043.049,E2 -2043.049} C_VEL
LIN {X 0,Y 573.544,Z 466.913,A -85,B 0,C 180,E1 -2043.825,E2 -2043.825} C_VEL
LIN {X 0,Y 573.421,Z 478.061,A -85,B 0,C 180,E1 -2044.743,E2 -2044.743} C_VEL
LIN {X 0,Y 573.304,Z 488.23,A -85,B 0,C 180,E1 -2045.754,E2 -2045.754} C_VEL
LIN {X 0,Y 573.2,Z 497.759,A -85,B 0,C 180,E1 -2046.9,E2 -2046.9} C_VEL
LIN {X 0,Y 573.101,Z 505.542,A -85,B 0,C 180,E1 -2048.037,E2 -2048.037} C_VEL
LIN {X 0,Y 573.034,Z 511.902,A -85,B 0,C 180,E1 -2049.166,E2 -2049.166} C_VEL
LIN {X 0,Y 573.035,Z 517.066,A -85,B 0,C 180,E1 -2050.29,E2 -2050.29} C_VEL
LIN {X 0,Y 572.995,Z 521.177,A -85,B 0,C 180,E1 -2051.404,E2 -2051.404} C_VEL
LIN {X 0,Y 572.965,Z 525.112,A -85,B 0,C 180,E1 -2052.88,E2 -2052.88} C_VEL
LIN {X 0,Y 572.93,Z 527.506,A -85,B 0,C 180,E1 -2054.344,E2 -2054.344} C_VEL
LIN {X 0,Y 572.973,Z 528.452,A -85,B 0,C 180,E1 -2055.8,E2 -2055.8} C_VEL
LIN {X 0,Y 572.942,Z 528.001,A -85,B 0,C 180,E1 -2057.245,E2 -2057.245} C_VEL
LIN {X 0,Y 572.96,Z 526.165,A -85,B 0,C 180,E1 -2058.682,E2 -2058.682} C_VEL
LIN {X 0,Y 572.976,Z 522.903,A -85,B 0,C 180,E1 -2060.112,E2 -2060.112} C_VEL
LIN {X 0,Y 573.016,Z 518.129,A -85,B 0,C 180,E1 -2061.537,E2 -2061.537} C_VEL
LIN {X 0,Y 573.055,Z 513.525,A -85,B 0,C 180,E1 -2062.602,E2 -2062.602} C_VEL
LIN {X 0,Y 573.111,Z 506.867,A -85,B 0,C 180,E1 -2063.841,E2 -2063.841} C_VEL
LIN {X 0,Y 573.19,Z 498.626,A -85,B 0,C 180,E1 -2065.077,E2 -2065.077} C_VEL
LIN {X 0,Y 573.278,Z 490.077,A -85,B 0,C 180,E1 -2066.134,E2 -2066.134} C_VEL
LIN {X 0,Y 573.432,Z 479.77,A -85,B 0,C 180,E1 -2067.19,E2 -2067.19} C_VEL
LIN {X 0,Y 573.525,Z 468.337,A -85,B 0,C 180,E1 -2068.157,E2 -2068.157} C_VEL
LIN {X 0,Y 573.728,Z 456.929,A -85,B 0,C 180,E1 -2068.947,E2 -2068.947} C_VEL
LIN {X 0,Y 573.882,Z 444.487,A -85,B 0,C 180,E1 -2069.649,E2 -2069.649} C_VEL
LIN {X 0,Y 574.042,Z 431.691,A -85,B 0,C 180,E1 -2070.219,E2 -2070.219} C_VEL
LIN {X 0,Y 574.137,Z 418.019,A -85,B 0,C 180,E1 -2070.68,E2 -2070.68} C_VEL
LIN {X 0,Y 574.225,Z 403.797,A -85,B 0,C 180,E1 -2071.008,E2 -2071.008} C_VEL
LIN {X 0,Y 574.493,Z 272.305,A -85,B 0,C 180,E1 -2072.695,E2 -2072.695} C_VEL
LIN {X 0,Y 573.457,Z 266.672,A -85,B 0,C 180,E1 -2072.81,E2 -2072.81} C_VEL
LIN {X 0,Y 573.699,Z 249.445,A -85,B 0,C 180,E1 -2075.448,E2 -2075.448} C_VEL
LIN {X 0,Y 573.67,Z 238.727,A -85,B 0,C 180,E1 -2077.116,E2 -2077.116} C_VEL
LIN {X 0,Y 573.283,Z 236.702,A -85,B 0,C 180,E1 -2077.484,E2 -2077.484} C_VEL
LIN {X 0,Y 573.226,Z 236.711,A -85,B 0,C 180,E1 -2079.883,E2 -2079.883} C_VEL
LIN {X 0,Y 573.266,Z 236.705,A -85,B 0,C 180,E1 -2082.029,E2 -2082.029} C_VEL
LIN {X 0,Y 573.227,Z 236.703,A -85,B 0,C 180,E1 -2084.92,E2 -2084.92} C_VEL
LIN {X 0,Y 573.245,Z 236.708,A -85,B 0,C 180,E1 -2087.848,E2 -2087.848} C_VEL
LIN {X 0,Y 573.245,Z 236.703,A -85,B 0,C 180,E1 -2090.077,E2 -2090.077} C_VEL
LIN {X 0,Y 573.228,Z 236.702,A -85,B 0,C 180,E1 -2092.338,E2 -2092.338} C_VEL
LIN {X 0,Y 573.247,Z 236.704,A -85,B 0,C 180,E1 -2095.41,E2 -2095.41} C_VEL
LIN {X 0,Y 573.252,Z 236.701,A -85,B 0,C 180,E1 -2098.032,E2 -2098.032} C_VEL
LIN {X 0,Y 573.231,Z 236.701,A -85,B 0,C 180,E1 -2100.886,E2 -2100.886} C_VEL
LIN {X 0,Y 573.274,Z 236.705,A -85,B 0,C 180,E1 -2103.528,E2 -2103.528} C_VEL
LIN {X 0,Y 573.247,Z 236.7,A -85,B 0,C 180,E1 -2106.048,E2 -2106.048} C_VEL
LIN {X 0,Y 573.236,Z 236.7,A -85,B 0,C 180,E1 -2108.701,E2 -2108.701} C_VEL
LIN {X 0,Y 573.252,Z 236.704,A -85,B 0,C 180,E1 -2111.598,E2 -2111.598} C_VEL
LIN {X 0,Y 573.224,Z 236.701,A -85,B 0,C 180,E1 -2114.333,E2 -2114.333} C_VEL
LIN {X 0,Y 573.246,Z 236.707,A -85,B 0,C 180,E1 -2117.357,E2 -2117.357} C_VEL
LIN {X 0,Y 573.238,Z 236.699,A -85,B 0,C 180,E1 -2120.394,E2 -2120.394} C_VEL
LIN {X 0,Y 573.244,Z 236.707,A -85,B 0,C 180,E1 -2123.079,E2 -2123.079} C_VEL
LIN {X 0,Y 573.264,Z 236.698,A -85,B 0,C 180,E1 -2125.673,E2 -2125.673} C_VEL
LIN {X 0,Y 573.237,Z 236.699,A -85,B 0,C 180,E1 -2128.186,E2 -2128.186} C_VEL
LIN {X 0,Y 573.258,Z 236.701,A -85,B 0,C 180,E1 -2130.635,E2 -2130.635} C_VEL
LIN {X 0,Y 573.262,Z 236.699,A -85,B 0,C 180,E1 -2133.5,E2 -2133.5} C_VEL
LIN {X 0,Y 573.223,Z 236.702,A -85,B 0,C 180,E1 -2136.136,E2 -2136.136} C_VEL
LIN {X 0,Y 573.25,Z 236.703,A -85,B 0,C 180,E1 -2139.175,E2 -2139.175} C_VEL
LIN {X 0,Y 573.228,Z 236.702,A -85,B 0,C 180,E1 -2141.413,E2 -2141.413} C_VEL
LIN {X 0,Y 573.25,Z 236.698,A -85,B 0,C 180,E1 -2143.623,E2 -2143.623} C_VEL
LIN {X 0,Y 573.231,Z 236.707,A -85,B 0,C 180,E1 -2146.531,E2 -2146.531} C_VEL
LIN {X 0,Y 573.251,Z 236.707,A -85,B 0,C 180,E1 -2148.746,E2 -2148.746} C_VEL
LIN {X 0,Y 573.282,Z 236.694,A -85,B 0,C 180,E1 -2151.542,E2 -2151.542} C_VEL
LIN {X 0,Y 573.286,Z 236.7,A -85,B 0,C 180,E1 -2154.373,E2 -2154.373} C_VEL
LIN {X 0,Y 573.301,Z 236.693,A -85,B 0,C 180,E1 -2157.893,E2 -2157.893} C_VEL
LIN {X 0,Y 573.328,Z 236.694,A -85,B 0,C 180,E1 -2160.703,E2 -2160.703} C_VEL
LIN {X 0,Y 573.232,Z 236.7,A -85,B 0,C 180,E1 -2163.515,E2 -2163.515} C_VEL
LIN {X 0,Y 573.287,Z 236.694,A -85,B 0,C 180,E1 -2165.629,E2 -2165.629} C_VEL
LIN {X 0,Y 573.284,Z 236.702,A -85,B 0,C 180,E1 -2168.46,E2 -2168.46} C_VEL
LIN {X 0,Y 573.264,Z 236.696,A -85,B 0,C 180,E1 -2171.313,E2 -2171.313} C_VEL
LIN {X 0,Y 573.267,Z 236.705,A -85,B 0,C 180,E1 -2174.194,E2 -2174.194} C_VEL
LIN {X 0,Y 573.253,Z 236.697,A -85,B 0,C 180,E1 -2177.112,E2 -2177.112} C_VEL
LIN {X 0,Y 573.248,Z 236.708,A -85,B 0,C 180,E1 -2180.077,E2 -2180.077} C_VEL
LIN {X 0,Y 573.228,Z 236.7,A -85,B 0,C 180,E1 -2183.1,E2 -2183.1} C_VEL
LIN {X 0,Y 573.25,Z 236.699,A -85,B 0,C 180,E1 -2185.411,E2 -2185.411} C_VEL
LIN {X 0,Y 573.259,Z 236.706,A -85,B 0,C 180,E1 -2188.032,E2 -2188.032} C_VEL
LIN {X 0,Y 573.239,Z 236.699,A -85,B 0,C 180,E1 -2190.886,E2 -2190.886} C_VEL
LIN {X 0,Y 573.258,Z 236.701,A -85,B 0,C 180,E1 -2193.525,E2 -2193.525} C_VEL
LIN {X 0,Y 573.258,Z 236.703,A -85,B 0,C 180,E1 -2196.049,E2 -2196.049} C_VEL
LIN {X 0,Y 573.246,Z 236.698,A -85,B 0,C 180,E1 -2198.702,E2 -2198.702} C_VEL
LIN {X 0,Y 573.227,Z 236.706,A -85,B 0,C 180,E1 -2201.458,E2 -2201.458} C_VEL
LIN {X 0,Y 573.233,Z 236.701,A -85,B 0,C 180,E1 -2204.334,E2 -2204.334} C_VEL
LIN {X 0,Y 573.243,Z 236.704,A -85,B 0,C 180,E1 -2207.359,E2 -2207.359} C_VEL
LIN {X 0,Y 573.238,Z 236.7,A -85,B 0,C 180,E1 -2210.393,E2 -2210.393} C_VEL
LIN {X 0,Y 573.251,Z 236.701,A -85,B 0,C 180,E1 -2213.078,E2 -2213.078} C_VEL
LIN {X 0,Y 573.268,Z 236.702,A -85,B 0,C 180,E1 -2215.672,E2 -2215.672} C_VEL
LIN {X 0,Y 573.244,Z 236.701,A -85,B 0,C 180,E1 -2218.185,E2 -2218.185} C_VEL
LIN {X 0,Y 573.264,Z 236.698,A -85,B 0,C 180,E1 -2220.635,E2 -2220.635} C_VEL
LIN {X 0,Y 573.252,Z 236.704,A -85,B 0,C 180,E1 -2223.025,E2 -2223.025} C_VEL
LIN {X 0,Y 573.304,Z 236.776,A -85,B 0,C 180,E1 -2225.44,E2 -2225.44} C_VEL
LIN {X 0,Y 574.26,Z 241.978,A -85,B 0,C 180,E1 -2226.18,E2 -2226.18} C_VEL
LIN {X 0,Y 574.02,Z 264.754,A -85,B 0,C 180,E1 -2229.203,E2 -2229.203} C_VEL
LIN {X 0,Y 573.721,Z 288.917,A -85,B 0,C 180,E1 -2232.37,E2 -2232.37} C_VEL
LIN {X 0,Y 573.634,Z 295.612,A -85,B 0,C 180,E1 -2233.237,E2 -2233.237} C_VEL
LIN {X 0,Y 574.592,Z 301.543,A -85,B 0,C 180,E1 -2233.343,E2 -2233.343} C_VEL
LIN {X 0,Y 574.277,Z 433.897,A -85,B 0,C 180,E1 -2235.04,E2 -2235.04} C_VEL
LIN {X 0,Y 574.135,Z 448.606,A -85,B 0,C 180,E1 -2235.383,E2 -2235.383} C_VEL
LIN {X 0,Y 573.995,Z 462.844,A -85,B 0,C 180,E1 -2235.871,E2 -2235.871} C_VEL
LIN {X 0,Y 573.873,Z 475.647,A -85,B 0,C 180,E1 -2236.455,E2 -2236.455} C_VEL
LIN {X 0,Y 573.711,Z 488.105,A -85,B 0,C 180,E1 -2237.172,E2 -2237.172} C_VEL
LIN {X 0,Y 573.532,Z 500.646,A -85,B 0,C 180,E1 -2238.066,E2 -2238.066} C_VEL
LIN {X 0,Y 573.45,Z 510.853,A -85,B 0,C 180,E1 -2238.955,E2 -2238.955} C_VEL
LIN {X 0,Y 573.269,Z 520.335,A -85,B 0,C 180,E1 -2239.939,E2 -2239.939} C_VEL
LIN {X 0,Y 573.197,Z 528.913,A -85,B 0,C 180,E1 -2241.006,E2 -2241.006} C_VEL
LIN {X 0,Y 573.112,Z 537.117,A -85,B 0,C 180,E1 -2242.248,E2 -2242.248} C_VEL
LIN {X 0,Y 573.036,Z 543.45,A -85,B 0,C 180,E1 -2243.427,E2 -2243.427} C_VEL
LIN {X 0,Y 573.001,Z 548.961,A -85,B 0,C 180,E1 -2244.722,E2 -2244.722} C_VEL
LIN {X 0,Y 573.028,Z 552.443,A -85,B 0,C 180,E1 -2245.78,E2 -2245.78} C_VEL
LIN {X 0,Y 572.956,Z 555.832,A -85,B 0,C 180,E1 -2247.188,E2 -2247.188} C_VEL
LIN {X 0,Y 572.941,Z 557.833,A -85,B 0,C 180,E1 -2248.594,E2 -2248.594} C_VEL
LIN {X 0,Y 572.937,Z 558.5,A -85,B 0,C 180,E1 -2250,E2 -2250} C_VEL
LIN {X 0,Y 572.941,Z 557.834,A -85,B 0,C 180,E1 -2251.406,E2 -2251.406} C_VEL
LIN {X 0,Y 572.956,Z 555.834,A -85,B 0,C 180,E1 -2252.812,E2 -2252.812} C_VEL
LIN {X 0,Y 573.028,Z 552.445,A -85,B 0,C 180,E1 -2254.22,E2 -2254.22} C_VEL
LIN {X 0,Y 573.057,Z 547.569,A -85,B 0,C 180,E1 -2255.63,E2 -2255.63} C_VEL
LIN {X 0,Y 573.065,Z 542.82,A -85,B 0,C 180,E1 -2256.699,E2 -2256.699} C_VEL
LIN {X 0,Y 573.126,Z 536.039,A -85,B 0,C 180,E1 -2257.929,E2 -2257.929} C_VEL
LIN {X 0,Y 573.225,Z 527.56,A -85,B 0,C 180,E1 -2259.171,E2 -2259.171} C_VEL
LIN {X 0,Y 573.304,Z 518.71,A -85,B 0,C 180,E1 -2260.239,E2 -2260.239} C_VEL
LIN {X 0,Y 573.462,Z 507.993,A -85,B 0,C 180,E1 -2261.308,E2 -2261.308} C_VEL
LIN {X 0,Y 573.62,Z 497.145,A -85,B 0,C 180,E1 -2262.201,E2 -2262.201} C_VEL
LIN {X 0,Y 573.764,Z 485.263,A -85,B 0,C 180,E1 -2263.007,E2 -2263.007} C_VEL
LIN {X 0,Y 573.937,Z 472.104,A -85,B 0,C 180,E1 -2263.724,E2 -2263.724} C_VEL
LIN {X 0,Y 574.119,Z 458.831,A -85,B 0,C 180,E1 -2264.283,E2 -2264.283} C_VEL
LIN {X 0,Y 574.204,Z 444.778,A -85,B 0,C 180,E1 -2264.721,E2 -2264.721} C_VEL
LIN {X 0,Y 574.27,Z 431.158,A -85,B 0,C 180,E1 -2265.005,E2 -2265.005} C_VEL
LIN {X 0,Y 574.522,Z 300.617,A -85,B 0,C 180,E1 -2266.671,E2 -2266.671} C_VEL
LIN {X 0,Y 573.616,Z 295.511,A -85,B 0,C 180,E1 -2266.776,E2 -2266.776} C_VEL
LIN {X 0,Y 573.852,Z 275.11,A -85,B 0,C 180,E1 -2269.434,E2 -2269.434} C_VEL
LIN {X 0,Y 574.134,Z 254.846,A -85,B 0,C 180,E1 -2272.111,E2 -2272.111} C_VEL
LIN {X 0,Y 574.231,Z 241.964,A -85,B 0,C 180,E1 -2273.821,E2 -2273.821} C_VEL
LIN {X 0,Y 573.298,Z 236.702,A -85,B 0,C 180,E1 -2274.584,E2 -2274.584} C_VEL
LIN {X 0,Y 573.251,Z 236.704,A -85,B 0,C 180,E1 -2276.975,E2 -2276.975} C_VEL
LIN {X 0,Y 573.247,Z 236.7,A -85,B 0,C 180,E1 -2279.487,E2 -2279.487} C_VEL
LIN {X 0,Y 573.255,Z 236.707,A -85,B 0,C 180,E1 -2282.644,E2 -2282.644} C_VEL
LIN {X 0,Y 573.207,Z 236.706,A -85,B 0,C 180,E1 -2285.187,E2 -2285.187} C_VEL
LIN {X 0,Y 573.233,Z 236.702,A -85,B 0,C 180,E1 -2287.807,E2 -2287.807} C_VEL
LIN {X 0,Y 573.242,Z 236.706,A -85,B 0,C 180,E1 -2290.524,E2 -2290.524} C_VEL
LIN {X 0,Y 573.245,Z 236.699,A -85,B 0,C 180,E1 -2293.357,E2 -2293.357} C_VEL
LIN {X 0,Y 573.241,Z 236.708,A -85,B 0,C 180,E1 -2296.33,E2 -2296.33} C_VEL
LIN {X 0,Y 573.27,Z 236.697,A -85,B 0,C 180,E1 -2299.476,E2 -2299.476} C_VEL
LIN {X 0,Y 573.233,Z 236.708,A -85,B 0,C 180,E1 -2302.192,E2 -2302.192} C_VEL
LIN {X 0,Y 573.264,Z 236.695,A -85,B 0,C 180,E1 -2304.816,E2 -2304.816} C_VEL
LIN {X 0,Y 573.25,Z 236.699,A -85,B 0,C 180,E1 -2307.354,E2 -2307.354} C_VEL
LIN {X 0,Y 573.251,Z 236.705,A -85,B 0,C 180,E1 -2309.823,E2 -2309.823} C_VEL
